LIN {X -0.120,Y -244.755,Z 514.218,A 0.000,B 0.000,C 90.000,E1 39.277} C_DIS
LIN {X -0.007,Y -235.366,Z 514.200,A 0.000,B 0.000,C 90.000,E1 35.931} C_DIS
LIN {X -0.130,Y -227.809,Z 514.183,A 0.000,B 0.000,C 90.000,E1 32.959} C_DIS
LIN {X 0.017,Y -221.054,Z 514.166,A 0.000,B 0.000,C 90.000,E1 29.873} C_DIS
LIN {X -0.038,Y -215.129,Z 514.149,A 0.000,B 0.000,C 90.000,E1 26.796} C_DIS
LIN {X 0.047,Y -210.062,Z 514.131,A 0.000,B 0.000,C 90.000,E1 23.643} C_DIS
LIN {X -0.028,Y -204.891,Z 514.109,A 0.000,B 0.000,C 90.000,E1 19.704} C_DIS
LIN {X -0.082,Y -200.758,Z 514.087,A 0.000,B 0.000,C 90.000,E1 15.717} C_DIS
LIN {X 0.030,Y -197.089,Z 514.060,A 0.000,B 0.000,C 90.000,E1 10.838} C_DIS
LIN {X -0.097,Y -194.452,Z 514.024,A 0.000,B 0.000,C 90.000,E1 4.359} C_DIS
LIN {X -0.009,Y -195.978,Z 513.961,A 0.000,B 0.000,C 90.000,E1 352.996} C_DIS
LIN {X 0.017,Y -199.614,Z 513.929,A 0.000,B 0.000,C 90.000,E1 347.297} C_DIS
LIN {X -0.001,Y -203.417,Z 513.907,A 0.000,B 0.000,C 90.000,E1 343.268} C_DIS
LIN {X 0.019,Y -208.024,Z 513.885,A 0.000,B 0.000,C 90.000,E1 339.263} C_DIS
LIN {X 0.017,Y -213.374,Z 513.863,A 0.000,B 0.000,C 90.000,E1 335.305} C_DIS
LIN {X 0.048,Y -219.357,Z 513.841,A 0.000,B 0.000,C 90.000,E1 331.385} C_DIS
LIN {X 0.009,Y -225.894,Z 513.820,A 0.000,B 0.000,C 90.000,E1 327.533} C_DIS
LIN {X 0.008,Y -231.651,Z 513.803,A 0.000,B 0.000,C 90.000,E1 324.482} C_DIS
LIN {X -0.005,Y -239.280,Z 513.782,A 0.000,B 0.000,C 90.000,E1 320.723} C_DIS
LIN {X -0.031,Y -247.836,Z 513.761,A 0.000,B 0.000,C 90.000,E1 317.025} C_DIS
LIN {X -0.010,Y -256.576,Z 513.743,A 0.000,B 0.000,C 90.000,E1 313.743} C_DIS
LIN {X 0.003,Y -267.396,Z 513.723,A 0.000,B 0.000,C 90.000,E1 310.172} C_DIS
LIN {X 0.088,Y -279.550,Z 513.704,A 0.000,B 0.000,C 90.000,E1 306.664} C_DIS
LIN {X -0.111,Y -292.992,Z 513.685,A 0.000,B 0.000,C 90.000,E1 303.293} C_DIS
LIN {X 0.095,Y -305.926,Z 513.668,A 0.000,B 0.000,C 90.000,E1 300.256} C_DIS
LIN {X 0.147,Y -321.556,Z 513.650,A 0.000,B 0.000,C 90.000,E1 297.001} C_DIS
LIN {X -0.195,Y -332.000,Z 513.640,A 0.000,B 0.000,C 90.000,E1 295.155} C_DIS
LIN {X -0.025,Y -349.412,Z 513.624,A 0.000,B 0.000,C 90.000,E1 292.333} C_DIS
LIN {X -0.077,Y -368.920,Z 513.609,A 0.000,B 0.000,C 90.000,E1 289.631} C_DIS
LIN {X 0.072,Y -390.367,Z 513.594,A 0.000,B 0.000,C 90.000,E1 286.985} C_DIS
LIN {X -0.161,Y -412.698,Z 513.580,A 0.000,B 0.000,C 90.000,E1 284.481} C_DIS
LIN {X 0.197,Y -425.211,Z 513.573,A 0.000,B 0.000,C 90.000,E1 283.063} C_DIS
LIN {X -0.216,Y -437.299,Z 513.565,A 0.000,B 0.000,C 90.000,E1 281.771} C_DIS
LIN {X 0.182,Y -446.567,Z 513.559,A 0.000,B 0.000,C 90.000,E1 280.658} C_DIS
LIN {X 0.176,Y -455.192,Z 513.554,A 0.000,B 0.000,C 90.000,E1 279.613} C_DIS
LIN {X -0.004,Y -461.099,Z 513.549,A 0.000,B 0.000,C 90.000,E1 278.859} C_DIS
LIN {X -0.140,Y -466.456,Z 513.545,A 0.000,B 0.000,C 90.000,E1 278.106} C_DIS
LIN {X 0.240,Y -471.291,Z 513.541,A 0.000,B 0.000,C 90.000,E1 277.296} C_DIS
LIN {X 0.136,Y -475.580,Z 513.536,A 0.000,B 0.000,C 90.000,E1 276.549} C_DIS
LIN {X 0.127,Y -479.382,Z 513.532,A 0.000,B 0.000,C 90.000,E1 275.796} C_DIS
LIN {X 0.096,Y -482.574,Z 513.528,A 0.000,B 0.000,C 90.000,E1 275.049} C_DIS
LIN {X -0.215,Y -484.338,Z 513.525,A 0.000,B 0.000,C 90.000,E1 274.588} C_DIS
LIN {X -0.075,Y -485.711,Z 513.523,A 0.000,B 0.000,C 90.000,E1 274.073} C_DIS
LIN {X 0.111,Y -486.806,Z 513.520,A 0.000,B 0.000,C 90.000,E1 273.555} C_DIS
LIN {X -0.185,Y -487.563,Z 513.517,A 0.000,B 0.000,C 90.000,E1 273.094} C_DIS
LIN {X -0.013,Y -487.993,Z 513.514,A 0.000,B 0.000,C 90.000,E1 272.579} C_DIS
LIN {X 0.165,Y -487.997,Z 513.512,A 0.000,B 0.000,C 90.000,E1 272.064} C_DIS
LIN {X -0.126,Y -487.649,Z 513.509,A 0.000,B 0.000,C 90.000,E1 271.604} C_DIS
LIN {X 0.056,Y -486.936,Z 513.506,A 0.000,B 0.000,C 90.000,E1 271.088} C_DIS
LIN {X 0.236,Y -485.739,Z 513.503,A 0.000,B 0.000,C 90.000,E1 270.573} C_DIS
LIN {X -0.073,Y -483.979,Z 513.501,A 0.000,B 0.000,C 90.000,E1 270.115} C_DIS
LIN {X 0.096,Y -481.572,Z 513.498,A 0.000,B 0.000,C 90.000,E1 269.599} C_DIS
LIN {X -0.232,Y -478.454,Z 513.495,A 0.000,B 0.000,C 90.000,E1 269.141} C_DIS
LIN {X -0.097,Y -474.407,Z 513.492,A 0.000,B 0.000,C 90.000,E1 268.625} C_DIS
LIN {X 0.195,Y -472.055,Z 513.491,A 0.000,B 0.000,C 90.000,E1 268.339} C_DIS
LIN {X -0.019,Y -466.542,Z 513.488,A 0.000,B 0.000,C 90.000,E1 267.879} C_DIS
LIN {X 0.146,Y -460.305,Z 513.486,A 0.000,B 0.000,C 90.000,E1 267.421} C_DIS
LIN {X -0.101,Y -456.798,Z 513.485,A 0.000,B 0.000,C 90.000,E1 267.249} C_DIS
LIN {X -0.038,Y -449.866,Z 513.483,A 0.000,B 0.000,C 90.000,E1 266.906} C_DIS
LIN {X 0.031,Y -442.828,Z 513.481,A 0.000,B 0.000,C 90.000,E1 266.617} C_DIS
LIN {X -0.015,Y -435.647,Z 513.480,A 0.000,B 0.000,C 90.000,E1 266.388} C_DIS
LIN {X -0.171,Y -427.820,Z 513.479,A 0.000,B 0.000,C 90.000,E1 266.216} C_DIS
LIN {X 0.052,Y -417.909,Z 513.478,A 0.000,B 0.000,C 90.000,E1 266.045} C_DIS
LIN {X 0.067,Y -409.310,Z 513.478,A 0.000,B 0.000,C 90.000,E1 265.988} C_DIS
LIN {X -0.005,Y -180.920,Z 513.478,A 0.000,B 0.000,C 90.000,E1 265.988} C_DIS
LIN {X -0.002,Y -180.885,Z 513.473,A 0.000,B 0.000,C 90.000,E1 265.122} C_DIS
LIN {X 0.056,Y -179.006,Z 513.445,A 0.000,B 0.000,C 90.000,E1 260.038} C_DIS
LIN {X -0.025,Y -178.614,Z 513.440,A 0.000,B 0.000,C 90.000,E1 259.218} C_DIS
LIN {X 0.043,Y -175.665,Z 513.412,A 0.000,B 0.000,C 90.000,E1 254.102} C_DIS
LIN {X 0.048,Y -172.383,Z 513.388,A 0.000,B 0.000,C 90.000,E1 249.826} C_DIS
LIN {X 0.062,Y -171.183,Z 513.378,A 0.000,B 0.000,C 90.000,E1 248.103} C_DIS
LIN {X -0.045,Y -167.476,Z 513.354,A 0.000,B 0.000,C 90.000,E1 243.819} C_DIS
LIN {X 0.039,Y -166.872,Z 513.350,A 0.000,B 0.000,C 90.000,E1 242.922} C_DIS
LIN {X -0.045,Y -162.177,Z 513.320,A 0.000,B 0.000,C 90.000,E1 237.709} C_DIS
LIN {X 0.013,Y -160.742,Z 513.311,A 0.000,B 0.000,C 90.000,E1 235.928} C_DIS
LIN {X -0.008,Y -157.542,Z 513.291,A 0.000,B 0.000,C 90.000,E1 232.396} C_DIS
LIN {X 0.048,Y -155.570,Z 513.276,A 0.000,B 0.000,C 90.000,E1 229.703} C_DIS
LIN {X -0.019,Y -151.857,Z 513.251,A 0.000,B 0.000,C 90.000,E1 225.243} C_DIS
LIN {X -0.004,Y -150.079,Z 513.236,A 0.000,B 0.000,C 90.000,E1 222.528} C_DIS
LIN {X 0.030,Y -146.884,Z 513.211,A 0.000,B 0.000,C 90.000,E1 217.971} C_DIS
LIN {X 0.019,Y -145.470,Z 513.196,A 0.000,B 0.000,C 90.000,E1 215.231} C_DIS
LIN {X -0.064,Y -142.882,Z 513.170,A 0.000,B 0.000,C 90.000,E1 210.669} C_DIS
LIN {X -0.007,Y -141.501,Z 513.150,A 0.000,B 0.000,C 90.000,E1 206.950} C_DIS
LIN {X 0.042,Y -139.388,Z 513.114,A 0.000,B 0.000,C 90.000,E1 200.429} C_DIS
LIN {X 0.030,Y -138.845,Z 513.098,A 0.000,B 0.000,C 90.000,E1 197.638} C_DIS
LIN {X -0.046,Y -138.353,Z 513.057,A 0.000,B 0.000,C 90.000,E1 190.197} C_DIS
LIN {X -0.054,Y -139.517,Z 513.005,A 0.000,B 0.000,C 90.000,E1 180.859} C_DIS
LIN {X 0.027,Y -141.172,Z 512.974,A 0.000,B 0.000,C 90.000,E1 175.241} C_DIS
LIN {X -0.002,Y -142.552,Z 512.958,A 0.000,B 0.000,C 90.000,E1 172.470} C_DIS
LIN {X -0.076,Y -144.830,Z 512.932,A 0.000,B 0.000,C 90.000,E1 167.881} C_DIS
LIN {X 0.052,Y -147.452,Z 512.912,A 0.000,B 0.000,C 90.000,E1 164.157} C_DIS
LIN {X -0.062,Y -150.033,Z 512.892,A 0.000,B 0.000,C 90.000,E1 160.550} C_DIS
LIN {X -0.056,Y -153.372,Z 512.872,A 0.000,B 0.000,C 90.000,E1 156.922} C_DIS
LIN {X -0.008,Y -155.905,Z 512.857,A 0.000,B 0.000,C 90.000,E1 154.204} C_DIS
LIN {X -0.032,Y -159.766,Z 512.837,A 0.000,B 0.000,C 90.000,E1 150.639} C_DIS
LIN {X -0.045,Y -162.006,Z 512.827,A 0.000,B 0.000,C 90.000,E1 148.869} C_DIS
LIN {X 0.069,Y -166.199,Z 512.807,A 0.000,B 0.000,C 90.000,E1 145.308} C_DIS
LIN {X 0.072,Y -171.215,Z 512.788,A 0.000,B 0.000,C 90.000,E1 141.823} C_DIS
LIN {X -0.005,Y -176.099,Z 512.769,A 0.000,B 0.000,C 90.000,E1 138.405} C_DIS
LIN {X 0.113,Y -180.362,Z 512.755,A 0.000,B 0.000,C 90.000,E1 135.810} C_DIS
LIN {X 0.090,Y -185.771,Z 512.736,A 0.000,B 0.000,C 90.000,E1 132.447} C_DIS
LIN {X 0.023,Y -190.385,Z 512.722,A 0.000,B 0.000,C 90.000,E1 129.967} C_DIS
LIN {X 0.020,Y -192.445,Z 512.715,A 0.000,B 0.000,C 90.000,E1 128.749} C_DIS
LIN {X -0.013,Y -289.228,Z 512.715,A 0.000,B 0.000,C 90.000,E1 128.749} C_DIS
LIN {X -0.057,Y -290.139,Z 512.715,A 0.000,B 0.000,C 90.000,E1 128.749} C_DIS
LIN {X -0.072,Y -295.347,Z 512.714,A 0.000,B 0.000,C 90.000,E1 128.543} C_DIS
LIN {X 0.100,Y -297.889,Z 512.713,A 0.000,B 0.000,C 90.000,E1 128.302} C_DIS
LIN {X 0.151,Y -301.704,Z 512.710,A 0.000,B 0.000,C 90.000,E1 127.810} C_DIS
LIN {X -0.090,Y -303.526,Z 512.708,A 0.000,B 0.000,C 90.000,E1 127.523} C_DIS
LIN {X 0.094,Y -304.951,Z 512.707,A 0.000,B 0.000,C 90.000,E1 127.156} C_DIS
LIN {X 0.071,Y -306.993,Z 512.703,A 0.000,B 0.000,C 90.000,E1 126.503} C_DIS
LIN {X 0.104,Y -317.017,Z 512.685,A 0.000,B 0.000,C 90.000,E1 123.245} C_DIS
LIN {X 0.027,Y -327.358,Z 512.669,A 0.000,B 0.000,C 90.000,E1 120.384} C_DIS
LIN {X -0.142,Y -339.055,Z 512.653,A 0.000,B 0.000,C 90.000,E1 117.590} C_DIS
LIN {X 0.187,Y -352.208,Z 512.638,A 0.000,B 0.000,C 90.000,E1 114.771} C_DIS
LIN {X 0.056,Y -365.222,Z 512.624,A 0.000,B 0.000,C 90.000,E1 112.386} C_DIS
LIN {X -0.172,Y -379.577,Z 512.611,A 0.000,B 0.000,C 90.000,E1 110.066} C_DIS
LIN {X -0.168,Y -395.376,Z 512.599,A 0.000,B 0.000,C 90.000,E1 107.764} C_DIS
LIN {X 0.109,Y -412.737,Z 512.586,A 0.000,B 0.000,C 90.000,E1 105.481} C_DIS
LIN {X 0.108,Y -431.774,Z 512.574,A 0.000,B 0.000,C 90.000,E1 103.300} C_DIS
LIN {X 0.167,Y -451.899,Z 512.563,A 0.000,B 0.000,C 90.000,E1 101.243} C_DIS
LIN {X 0.055,Y -472.572,Z 512.552,A 0.000,B 0.000,C 90.000,E1 99.378} C_DIS
LIN {X 0.192,Y -477.818,Z 512.550,A 0.000,B 0.000,C 90.000,E1 98.916} C_DIS
LIN {X -0.229,Y -480.089,Z 512.548,A 0.000,B 0.000,C 90.000,E1 98.746} C_DIS
LIN {X 0.198,Y -481.950,Z 512.547,A 0.000,B 0.000,C 90.000,E1 98.454} C_DIS
LIN {X 0.149,Y -483.362,Z 512.546,A 0.000,B 0.000,C 90.000,E1 98.219} C_DIS
LIN {X -0.159,Y -485.241,Z 512.543,A 0.000,B 0.000,C 90.000,E1 97.757} C_DIS
LIN {X 0.023,Y -486.010,Z 512.540,A 0.000,B 0.000,C 90.000,E1 97.239} C_DIS
LIN {X 0.218,Y -485.794,Z 512.537,A 0.000,B 0.000,C 90.000,E1 96.720} C_DIS
LIN {X -0.066,Y -484.563,Z 512.535,A 0.000,B 0.000,C 90.000,E1 96.258} C_DIS
LIN {X -0.182,Y -483.507,Z 512.533,A 0.000,B 0.000,C 90.000,E1 96.024} C_DIS
LIN {X 0.131,Y -482.084,Z 512.532,A 0.000,B 0.000,C 90.000,E1 95.739} C_DIS
LIN {X -0.005,Y -474.162,Z 512.526,A 0.000,B 0.000,C 90.000,E1 94.759} C_DIS
LIN {X 0.071,Y -460.399,Z 512.517,A 0.000,B 0.000,C 90.000,E1 92.980} C_DIS
LIN {X -0.110,Y -451.472,Z 512.509,A 0.000,B 0.000,C 90.000,E1 91.718} C_DIS
LIN {X -0.135,Y -436.900,Z 512.496,A 0.000,B 0.000,C 90.000,E1 89.370} C_DIS
LIN {X 0.203,Y -423.873,Z 512.485,A 0.000,B 0.000,C 90.000,E1 87.192} C_DIS
LIN {X -0.138,Y -411.086,Z 512.472,A 0.000,B 0.000,C 90.000,E1 85.065} C_DIS
LIN {X 0.117,Y -397.019,Z 512.459,A 0.000,B 0.000,C 90.000,E1 82.534} C_DIS
LIN {X 0.107,Y -386.038,Z 512.448,A 0.000,B 0.000,C 90.000,E1 80.557} C_DIS
LIN {X -0.111,Y -375.042,Z 512.436,A 0.000,B 0.000,C 90.000,E1 78.578} C_DIS
LIN {X -0.045,Y -364.309,Z 512.425,A 0.000,B 0.000,C 90.000,E1 76.520} C_DIS
LIN {X -0.165,Y -353.218,Z 512.412,A 0.000,B 0.000,C 90.000,E1 74.157} C_DIS
LIN {X 0.067,Y -344.586,Z 512.400,A 0.000,B 0.000,C 90.000,E1 72.000} C_DIS
LIN {X -0.120,Y -333.650,Z 512.383,A 0.000,B 0.000,C 90.000,E1 68.954} C_DIS
LIN {X -0.035,Y -321.585,Z 512.362,A 0.000,B 0.000,C 90.000,E1 65.177} C_DIS
LIN {X 0.020,Y -313.768,Z 512.348,A 0.000,B 0.000,C 90.000,E1 62.615} C_DIS
LIN {X 0.077,Y -307.963,Z 512.337,A 0.000,B 0.000,C 90.000,E1 60.667} C_DIS
LIN {X -0.032,Y -300.214,Z 512.323,A 0.000,B 0.000,C 90.000,E1 58.074} C_DIS
LIN {X -0.101,Y -290.942,Z 512.304,A 0.000,B 0.000,C 90.000,E1 54.769} C_DIS
LIN {X -0.055,Y -283.932,Z 512.289,A 0.000,B 0.000,C 90.000,E1 52.065} C_DIS
LIN {X -0.147,Y -280.320,Z 512.282,A 0.000,B 0.000,C 90.000,E1 50.723} C_DIS
LIN {X -0.061,Y -274.511,Z 512.270,A 0.000,B 0.000,C 90.000,E1 48.647} C_DIS
LIN {X -0.018,Y -269.212,Z 512.261,A 0.000,B 0.000,C 90.000,E1 46.905} C_DIS
LIN {X -0.009,Y -262.316,Z 512.249,A 0.000,B 0.000,C 90.000,E1 44.798} C_DIS
LIN {X -0.058,Y -251.867,Z 512.231,A 0.000,B 0.000,C 90.000,E1 41.595} C_DIS
LIN {X 0.008,Y -242.993,Z 512.215,A 0.000,B 0.000,C 90.000,E1 38.669} C_DIS
LIN {X -0.042,Y -234.757,Z 512.198,A 0.000,B 0.000,C 90.000,E1 35.724} C_DIS
LIN {X 0.014,Y -227.236,Z 512.182,A 0.000,B 0.000,C 90.000,E1 32.704} C_DIS
LIN {X -0.045,Y -220.548,Z 512.165,A 0.000,B 0.000,C 90.000,E1 29.667} C_DIS
LIN {X -0.019,Y -214.687,Z 512.148,A 0.000,B 0.000,C 90.000,E1 26.565} C_DIS
LIN {X -0.045,Y -209.696,Z 512.130,A 0.000,B 0.000,C 90.000,E1 23.439} C_DIS
LIN {X 0.055,Y -204.595,Z 512.108,A 0.000,B 0.000,C 90.000,E1 19.450} C_DIS
LIN {X -0.074,Y -200.511,Z 512.086,A 0.000,B 0.000,C 90.000,E1 15.481} C_DIS
LIN {X 0.028,Y -196.901,Z 512.059,A 0.000,B 0.000,C 90.000,E1 10.602} C_DIS
LIN {X 0.063,Y -194.347,Z 512.023,A 0.000,B 0.000,C 90.000,E1 4.073} C_DIS
LIN {X -0.014,Y -195.866,Z 511.961,A 0.000,B 0.000,C 90.000,E1 352.996} C_DIS
LIN {X 0.006,Y -199.485,Z 511.929,A 0.000,B 0.000,C 90.000,E1 347.297} C_DIS
LIN {X -0.016,Y -203.277,Z 511.907,A 0.000,B 0.000,C 90.000,E1 343.268} C_DIS
LIN {X -0.001,Y -207.891,Z 511.885,A 0.000,B 0.000,C 90.000,E1 339.263} C_DIS
LIN {X -0.007,Y -213.248,Z 511.863,A 0.000,B 0.000,C 90.000,E1 335.305} C_DIS
LIN {X 0.019,Y -219.221,Z 511.841,A 0.000,B 0.000,C 90.000,E1 331.385} C_DIS
LIN {X -0.026,Y -225.768,Z 511.820,A 0.000,B 0.000,C 90.000,E1 327.533} C_DIS
LIN {X -0.030,Y -231.544,Z 511.803,A 0.000,B 0.000,C 90.000,E1 324.482} C_DIS
LIN {X -0.047,Y -239.189,Z 511.782,A 0.000,B 0.000,C 90.000,E1 320.723} C_DIS
LIN {X 0.091,Y -247.765,Z 511.761,A 0.000,B 0.000,C 90.000,E1 316.986} C_DIS
LIN {X -0.048,Y -257.577,Z 511.741,A 0.000,B 0.000,C 90.000,E1 313.380} C_DIS
LIN {X 0.013,Y -268.530,Z 511.721,A 0.000,B 0.000,C 90.000,E1 309.806} C_DIS
LIN {X 0.135,Y -280.829,Z 511.702,A 0.000,B 0.000,C 90.000,E1 306.297} C_DIS
LIN {X -0.188,Y -294.405,Z 511.683,A 0.000,B 0.000,C 90.000,E1 302.959} C_DIS
LIN {X -0.060,Y -308.915,Z 511.664,A 0.000,B 0.000,C 90.000,E1 299.617} C_DIS
LIN {X 0.014,Y -323.243,Z 511.648,A 0.000,B 0.000,C 90.000,E1 296.693} C_DIS
LIN {X 0.146,Y -333.874,Z 511.638,A 0.000,B 0.000,C 90.000,E1 294.771} C_DIS
LIN {X -0.095,Y -349.446,Z 511.624,A 0.000,B 0.000,C 90.000,E1 292.333} C_DIS
LIN {X -0.152,Y -368.953,Z 511.609,A 0.000,B 0.000,C 90.000,E1 289.631} C_DIS
LIN {X -0.005,Y -390.388,Z 511.594,A 0.000,B 0.000,C 90.000,E1 286.985} C_DIS
LIN {X -0.197,Y -412.721,Z 511.580,A 0.000,B 0.000,C 90.000,E1 284.481} C_DIS
LIN {X -0.138,Y -425.120,Z 511.573,A 0.000,B 0.000,C 90.000,E1 283.119} C_DIS
LIN {X -0.135,Y -437.238,Z 511.565,A 0.000,B 0.000,C 90.000,E1 281.771} C_DIS
LIN {X -0.175,Y -446.550,Z 511.559,A 0.000,B 0.000,C 90.000,E1 280.715} C_DIS
LIN {X 0.011,Y -453.120,Z 511.555,A 0.000,B 0.000,C 90.000,E1 279.905} C_DIS
LIN {X -0.194,Y -459.252,Z 511.551,A 0.000,B 0.000,C 90.000,E1 279.151} C_DIS
LIN {X 0.119,Y -464.777,Z 511.546,A 0.000,B 0.000,C 90.000,E1 278.341} C_DIS
LIN {X 0.017,Y -469.791,Z 511.542,A 0.000,B 0.000,C 90.000,E1 277.587} C_DIS
LIN {X -0.041,Y -474.245,Z 511.538,A 0.000,B 0.000,C 90.000,E1 276.834} C_DIS
LIN {X -0.119,Y -478.215,Z 511.534,A 0.000,B 0.000,C 90.000,E1 276.087} C_DIS
LIN {X -0.111,Y -481.656,Z 511.530,A 0.000,B 0.000,C 90.000,E1 275.334} C_DIS
LIN {X -0.124,Y -484.402,Z 511.525,A 0.000,B 0.000,C 90.000,E1 274.588} C_DIS
LIN {X 0.017,Y -485.820,Z 511.523,A 0.000,B 0.000,C 90.000,E1 274.073} C_DIS
LIN {X 0.204,Y -486.894,Z 511.520,A 0.000,B 0.000,C 90.000,E1 273.555} C_DIS
LIN {X -0.091,Y -487.670,Z 511.517,A 0.000,B 0.000,C 90.000,E1 273.094} C_DIS
LIN {X 0.080,Y -488.091,Z 511.514,A 0.000,B 0.000,C 90.000,E1 272.579} C_DIS
LIN {X -0.228,Y -488.143,Z 511.512,A 0.000,B 0.000,C 90.000,E1 272.121} C_DIS
LIN {X -0.030,Y -487.800,Z 511.509,A 0.000,B 0.000,C 90.000,E1 271.604} C_DIS
LIN {X 0.152,Y -487.051,Z 511.506,A 0.000,B 0.000,C 90.000,E1 271.088} C_DIS
LIN {X -0.153,Y -485.877,Z 511.503,A 0.000,B 0.000,C 90.000,E1 270.630} C_DIS
LIN {X 0.024,Y -484.136,Z 511.501,A 0.000,B 0.000,C 90.000,E1 270.115} C_DIS
LIN {X 0.193,Y -481.736,Z 511.498,A 0.000,B 0.000,C 90.000,E1 269.599} C_DIS
LIN {X -0.135,Y -478.606,Z 511.495,A 0.000,B 0.000,C 90.000,E1 269.141} C_DIS
LIN {X 0.001,Y -474.582,Z 511.492,A 0.000,B 0.000,C 90.000,E1 268.625} C_DIS
LIN {X -0.180,Y -472.222,Z 511.491,A 0.000,B 0.000,C 90.000,E1 268.396} C_DIS
LIN {X 0.054,Y -466.727,Z 511.488,A 0.000,B 0.000,C 90.000,E1 267.879} C_DIS
LIN {X 0.189,Y -460.442,Z 511.486,A 0.000,B 0.000,C 90.000,E1 267.421} C_DIS
LIN {X -0.028,Y -453.674,Z 511.484,A 0.000,B 0.000,C 90.000,E1 267.078} C_DIS
LIN {X -0.160,Y -446.790,Z 511.482,A 0.000,B 0.000,C 90.000,E1 266.788} C_DIS
LIN {X 0.047,Y -439.832,Z 511.481,A 0.000,B 0.000,C 90.000,E1 266.502} C_DIS
LIN {X 0.133,Y -432.419,Z 511.479,A 0.000,B 0.000,C 90.000,E1 266.274} C_DIS
LIN {X 0.152,Y -423.889,Z 511.478,A 0.000,B 0.000,C 90.000,E1 266.102} C_DIS
LIN {X 0.044,Y -418.120,Z 511.478,A 0.000,B 0.000,C 90.000,E1 266.045} C_DIS
LIN {X 0.058,Y -410.283,Z 511.478,A 0.000,B 0.000,C 90.000,E1 265.988} C_DIS
LIN {X -0.009,Y -180.919,Z 511.478,A 0.000,B 0.000,C 90.000,E1 265.988} C_DIS
LIN {X -0.007,Y -180.885,Z 511.473,A 0.000,B 0.000,C 90.000,E1 265.122} C_DIS
LIN {X 0.052,Y -179.006,Z 511.445,A 0.000,B 0.000,C 90.000,E1 260.038} C_DIS
LIN {X -0.029,Y -178.612,Z 511.440,A 0.000,B 0.000,C 90.000,E1 259.218} C_DIS
LIN {X 0.039,Y -175.664,Z 511.412,A 0.000,B 0.000,C 90.000,E1 254.102} C_DIS
LIN {X 0.044,Y -172.382,Z 511.388,A 0.000,B 0.000,C 90.000,E1 249.826} C_DIS
LIN {X 0.058,Y -171.181,Z 511.378,A 0.000,B 0.000,C 90.000,E1 248.103} C_DIS
LIN {X -0.049,Y -167.475,Z 511.354,A 0.000,B 0.000,C 90.000,E1 243.819} C_DIS
LIN {X 0.034,Y -166.871,Z 511.350,A 0.000,B 0.000,C 90.000,E1 242.922} C_DIS
LIN {X -0.049,Y -162.176,Z 511.320,A 0.000,B 0.000,C 90.000,E1 237.709} C_DIS
LIN {X 0.008,Y -160.741,Z 511.311,A 0.000,B 0.000,C 90.000,E1 235.928} C_DIS
LIN {X -0.013,Y -157.542,Z 511.291,A 0.000,B 0.000,C 90.000,E1 232.396} C_DIS
LIN {X 0.045,Y -155.569,Z 511.276,A 0.000,B 0.000,C 90.000,E1 229.703} C_DIS
LIN {X -0.022,Y -151.857,Z 511.251,A 0.000,B 0.000,C 90.000,E1 225.243} C_DIS
LIN {X -0.008,Y -150.078,Z 511.236,A 0.000,B 0.000,C 90.000,E1 222.528} C_DIS
LIN {X 0.026,Y -146.883,Z 511.211,A 0.000,B 0.000,C 90.000,E1 217.971} C_DIS
LIN {X 0.015,Y -145.469,Z 511.196,A 0.000,B 0.000,C 90.000,E1 215.231} C_DIS
LIN {X -0.068,Y -142.881,Z 511.170,A 0.000,B 0.000,C 90.000,E1 210.669} C_DIS
LIN {X -0.011,Y -141.500,Z 511.150,A 0.000,B 0.000,C 90.000,E1 206.950} C_DIS
LIN {X 0.038,Y -139.387,Z 511.114,A 0.000,B 0.000,C 90.000,E1 200.429} C_DIS
LIN {X 0.027,Y -138.845,Z 511.098,A 0.000,B 0.000,C 90.000,E1 197.638} C_DIS
LIN {X -0.049,Y -138.354,Z 511.057,A 0.000,B 0.000,C 90.000,E1 190.197} C_DIS
LIN {X -0.058,Y -139.517,Z 511.005,A 0.000,B 0.000,C 90.000,E1 180.859} C_DIS
LIN {X 0.023,Y -141.174,Z 510.974,A 0.000,B 0.000,C 90.000,E1 175.241} C_DIS
LIN {X -0.006,Y -142.552,Z 510.958,A 0.000,B 0.000,C 90.000,E1 172.470} C_DIS
LIN {X -0.080,Y -144.830,Z 510.932,A 0.000,B 0.000,C 90.000,E1 167.881} C_DIS
LIN {X 0.048,Y -147.453,Z 510.912,A 0.000,B 0.000,C 90.000,E1 164.157} C_DIS
LIN {X -0.066,Y -150.035,Z 510.892,A 0.000,B 0.000,C 90.000,E1 160.550} C_DIS
LIN {X -0.060,Y -153.374,Z 510.872,A 0.000,B 0.000,C 90.000,E1 156.922} C_DIS
LIN {X -0.012,Y -155.906,Z 510.857,A 0.000,B 0.000,C 90.000,E1 154.204} C_DIS
LIN {X 0.103,Y -159.768,Z 510.837,A 0.000,B 0.000,C 90.000,E1 150.589} C_DIS
LIN {X -0.049,Y -162.008,Z 510.827,A 0.000,B 0.000,C 90.000,E1 148.869} C_DIS
LIN {X 0.064,Y -166.201,Z 510.807,A 0.000,B 0.000,C 90.000,E1 145.308} C_DIS
LIN {X 0.067,Y -171.217,Z 510.788,A 0.000,B 0.000,C 90.000,E1 141.823} C_DIS
LIN {X -0.009,Y -176.102,Z 510.769,A 0.000,B 0.000,C 90.000,E1 138.405} C_DIS
LIN {X 0.108,Y -180.364,Z 510.755,A 0.000,B 0.000,C 90.000,E1 135.810} C_DIS
LIN {X 0.086,Y -185.773,Z 510.736,A 0.000,B 0.000,C 90.000,E1 132.447} C_DIS
LIN {X 0.018,Y -190.388,Z 510.722,A 0.000,B 0.000,C 90.000,E1 129.967} C_DIS
LIN {X -0.091,Y -192.501,Z 510.715,A 0.000,B 0.000,C 90.000,E1 128.749} C_DIS
LIN {X 0.055,Y -289.106,Z 510.715,A 0.000,B 0.000,C 90.000,E1 128.705} C_DIS
LIN {X 0.063,Y -291.444,Z 510.715,A 0.000,B 0.000,C 90.000,E1 128.669} C_DIS
LIN {X -0.038,Y -295.372,Z 510.714,A 0.000,B 0.000,C 90.000,E1 128.508} C_DIS
LIN {X 0.093,Y -297.636,Z 510.713,A 0.000,B 0.000,C 90.000,E1 128.302} C_DIS
LIN {X -0.035,Y -301.507,Z 510.710,A 0.000,B 0.000,C 90.000,E1 127.855} C_DIS
LIN {X -0.020,Y -303.372,Z 510.708,A 0.000,B 0.000,C 90.000,E1 127.523} C_DIS
LIN {X 0.181,Y -304.833,Z 510.707,A 0.000,B 0.000,C 90.000,E1 127.156} C_DIS
LIN {X 0.159,Y -306.927,Z 510.703,A 0.000,B 0.000,C 90.000,E1 126.503} C_DIS
LIN {X -0.074,Y -316.942,Z 510.685,A 0.000,B 0.000,C 90.000,E1 123.293} C_DIS
LIN {X -0.050,Y -327.277,Z 510.669,A 0.000,B 0.000,C 90.000,E1 120.413} C_DIS
LIN {X -0.053,Y -338.966,Z 510.653,A 0.000,B 0.000,C 90.000,E1 117.590} C_DIS
LIN {X -0.042,Y -352.110,Z 510.638,A 0.000,B 0.000,C 90.000,E1 114.823} C_DIS
LIN {X 0.008,Y -365.117,Z 510.625,A 0.000,B 0.000,C 90.000,E1 112.408} C_DIS
LIN {X -0.080,Y -379.461,Z 510.611,A 0.000,B 0.000,C 90.000,E1 110.066} C_DIS
LIN {X -0.075,Y -395.253,Z 510.599,A 0.000,B 0.000,C 90.000,E1 107.764} C_DIS
LIN {X 0.204,Y -412.603,Z 510.586,A 0.000,B 0.000,C 90.000,E1 105.481} C_DIS
LIN {X 0.201,Y -431.630,Z 510.574,A 0.000,B 0.000,C 90.000,E1 103.300} C_DIS
LIN {X -0.187,Y -451.753,Z 510.563,A 0.000,B 0.000,C 90.000,E1 101.299} C_DIS
LIN {X 0.139,Y -472.423,Z 510.552,A 0.000,B 0.000,C 90.000,E1 99.378} C_DIS
LIN {X -0.196,Y -477.668,Z 510.550,A 0.000,B 0.000,C 90.000,E1 98.973} C_DIS
LIN {X -0.146,Y -480.018,Z 510.548,A 0.000,B 0.000,C 90.000,E1 98.746} C_DIS
LIN {X -0.154,Y -481.904,Z 510.547,A 0.000,B 0.000,C 90.000,E1 98.511} C_DIS
LIN {X -0.164,Y -483.342,Z 510.546,A 0.000,B 0.000,C 90.000,E1 98.276} C_DIS
LIN {X 0.008,Y -485.313,Z 510.543,A 0.000,B 0.000,C 90.000,E1 97.757} C_DIS
LIN {X 0.190,Y -486.155,Z 510.540,A 0.000,B 0.000,C 90.000,E1 97.239} C_DIS
LIN {X -0.098,Y -486.009,Z 510.538,A 0.000,B 0.000,C 90.000,E1 96.777} C_DIS
LIN {X 0.102,Y -484.856,Z 510.535,A 0.000,B 0.000,C 90.000,E1 96.258} C_DIS
LIN {X -0.065,Y -483.846,Z 510.533,A 0.000,B 0.000,C 90.000,E1 96.030} C_DIS
LIN {X -0.181,Y -482.481,Z 510.532,A 0.000,B 0.000,C 90.000,E1 95.796} C_DIS
LIN {X 0.003,Y -478.668,Z 510.529,A 0.000,B 0.000,C 90.000,E1 95.277} C_DIS
LIN {X -0.216,Y -460.814,Z 510.517,A 0.000,B 0.000,C 90.000,E1 93.037} C_DIS
LIN {X 0.065,Y -451.837,Z 510.510,A 0.000,B 0.000,C 90.000,E1 91.718} C_DIS
LIN {X 0.043,Y -437.213,Z 510.497,A 0.000,B 0.000,C 90.000,E1 89.370} C_DIS
LIN {X -0.040,Y -424.180,Z 510.485,A 0.000,B 0.000,C 90.000,E1 87.249} C_DIS
LIN {X 0.045,Y -411.362,Z 510.473,A 0.000,B 0.000,C 90.000,E1 85.065} C_DIS
LIN {X -0.093,Y -397.286,Z 510.459,A 0.000,B 0.000,C 90.000,E1 82.591} C_DIS
LIN {X -0.152,Y -386.312,Z 510.448,A 0.000,B 0.000,C 90.000,E1 80.622} C_DIS
LIN {X 0.074,Y -375.305,Z 510.437,A 0.000,B 0.000,C 90.000,E1 78.578} C_DIS
LIN {X 0.055,Y -364.562,Z 510.425,A 0.000,B 0.000,C 90.000,E1 76.533} C_DIS
LIN {X 0.021,Y -353.443,Z 510.412,A 0.000,B 0.000,C 90.000,E1 74.157} C_DIS
LIN {X -0.099,Y -345.947,Z 510.402,A 0.000,B 0.000,C 90.000,E1 72.362} C_DIS
LIN {X 0.034,Y -331.676,Z 510.380,A 0.000,B 0.000,C 90.000,E1 68.337} C_DIS
LIN {X -0.150,Y -321.683,Z 510.362,A 0.000,B 0.000,C 90.000,E1 65.229} C_DIS
LIN {X -0.085,Y -313.862,Z 510.348,A 0.000,B 0.000,C 90.000,E1 62.666} C_DIS
LIN {X -0.018,Y -308.033,Z 510.337,A 0.000,B 0.000,C 90.000,E1 60.717} C_DIS
LIN {X -0.116,Y -300.256,Z 510.323,A 0.000,B 0.000,C 90.000,E1 58.122} C_DIS
LIN {X 0.066,Y -290.958,Z 510.304,A 0.000,B 0.000,C 90.000,E1 54.769} C_DIS
LIN {X -0.117,Y -283.934,Z 510.289,A 0.000,B 0.000,C 90.000,E1 52.110} C_DIS
LIN {X 0.013,Y -280.329,Z 510.282,A 0.000,B 0.000,C 90.000,E1 50.723} C_DIS
LIN {X -0.110,Y -274.531,Z 510.270,A 0.000,B 0.000,C 90.000,E1 48.690} C_DIS
LIN {X -0.047,Y -269.231,Z 510.261,A 0.000,B 0.000,C 90.000,E1 46.944} C_DIS
LIN {X -0.044,Y -262.323,Z 510.249,A 0.000,B 0.000,C 90.000,E1 44.838} C_DIS
LIN {X -0.109,Y -253.025,Z 510.233,A 0.000,B 0.000,C 90.000,E1 42.000} C_DIS
LIN {X -0.002,Y -243.046,Z 510.215,A 0.000,B 0.000,C 90.000,E1 38.705} C_DIS
LIN {X 0.096,Y -234.808,Z 510.199,A 0.000,B 0.000,C 90.000,E1 35.724} C_DIS
LIN {X -0.044,Y -227.258,Z 510.182,A 0.000,B 0.000,C 90.000,E1 32.752} C_DIS
LIN {X 0.086,Y -220.569,Z 510.165,A 0.000,B 0.000,C 90.000,E1 29.667} C_DIS
LIN {X -0.084,Y -214.699,Z 510.148,A 0.000,B 0.000,C 90.000,E1 26.616} C_DIS
LIN {X -0.003,Y -209.715,Z 510.130,A 0.000,B 0.000,C 90.000,E1 23.462} C_DIS
LIN {X -0.017,Y -204.611,Z 510.108,A 0.000,B 0.000,C 90.000,E1 19.504} C_DIS
LIN {X 0.047,Y -200.500,Z 510.086,A 0.000,B 0.000,C 90.000,E1 15.481} C_DIS
LIN {X -0.048,Y -196.878,Z 510.059,A 0.000,B 0.000,C 90.000,E1 10.658} C_DIS
LIN {X -0.017,Y -194.290,Z 510.023,A 0.000,B 0.000,C 90.000,E1 4.131} C_DIS
LIN {X -0.019,Y -195.756,Z 509.961,A 0.000,B 0.000,C 90.000,E1 352.996} C_DIS
LIN {X -0.004,Y -199.355,Z 509.929,A 0.000,B 0.000,C 90.000,E1 347.297} C_DIS
LIN {X -0.030,Y -203.138,Z 509.907,A 0.000,B 0.000,C 90.000,E1 343.268} C_DIS
LIN {X -0.020,Y -207.755,Z 509.885,A 0.000,B 0.000,C 90.000,E1 339.263} C_DIS
LIN {X 0.058,Y -213.135,Z 509.863,A 0.000,B 0.000,C 90.000,E1 335.281} C_DIS
LIN {X -0.011,Y -219.085,Z 509.841,A 0.000,B 0.000,C 90.000,E1 331.385} C_DIS
LIN {X -0.060,Y -225.647,Z 509.820,A 0.000,B 0.000,C 90.000,E1 327.533} C_DIS
LIN {X 0.020,Y -232.922,Z 509.798,A 0.000,B 0.000,C 90.000,E1 323.703} C_DIS
LIN {X -0.143,Y -240.718,Z 509.778,A 0.000,B 0.000,C 90.000,E1 319.989} C_DIS
LIN {X -0.148,Y -249.548,Z 509.757,A 0.000,B 0.000,C 90.000,E1 316.296} C_DIS
LIN {X -0.070,Y -258.590,Z 509.739,A 0.000,B 0.000,C 90.000,E1 313.014} C_DIS
LIN {X 0.029,Y -269.675,Z 509.719,A 0.000,B 0.000,C 90.000,E1 309.439} C_DIS
LIN {X 0.023,Y -282.122,Z 509.700,A 0.000,B 0.000,C 90.000,E1 305.964} C_DIS
LIN {X 0.152,Y -295.814,Z 509.681,A 0.000,B 0.000,C 90.000,E1 302.546} C_DIS
LIN {X -0.084,Y -310.467,Z 509.663,A 0.000,B 0.000,C 90.000,E1 299.283} C_DIS
LIN {X -0.053,Y -323.264,Z 509.648,A 0.000,B 0.000,C 90.000,E1 296.693} C_DIS
LIN {X 0.077,Y -333.898,Z 509.638,A 0.000,B 0.000,C 90.000,E1 294.771} C_DIS
LIN {X -0.167,Y -349.480,Z 509.624,A 0.000,B 0.000,C 90.000,E1 292.333} C_DIS
LIN {X 0.121,Y -368.990,Z 509.609,A 0.000,B 0.000,C 90.000,E1 289.577} C_DIS
LIN {X -0.109,Y -387.983,Z 509.596,A 0.000,B 0.000,C 90.000,E1 287.275} C_DIS
LIN {X -0.215,Y -412.715,Z 509.580,A 0.000,B 0.000,C 90.000,E1 284.481} C_DIS
LIN {X -0.164,Y -425.156,Z 509.573,A 0.000,B 0.000,C 90.000,E1 283.119} C_DIS
LIN {X -0.158,Y -437.311,Z 509.565,A 0.000,B 0.000,C 90.000,E1 281.771} C_DIS
LIN {X 0.241,Y -446.663,Z 509.559,A 0.000,B 0.000,C 90.000,E1 280.658} C_DIS
LIN {X -0.213,Y -455.339,Z 509.554,A 0.000,B 0.000,C 90.000,E1 279.670} C_DIS
LIN {X 0.059,Y -461.301,Z 509.549,A 0.000,B 0.000,C 90.000,E1 278.859} C_DIS
LIN {X -0.075,Y -466.657,Z 509.545,A 0.000,B 0.000,C 90.000,E1 278.106} C_DIS
LIN {X -0.160,Y -471.479,Z 509.541,A 0.000,B 0.000,C 90.000,E1 277.352} C_DIS
LIN {X 0.206,Y -475.771,Z 509.537,A 0.000,B 0.000,C 90.000,E1 276.549} C_DIS
LIN {X 0.198,Y -479.526,Z 509.532,A 0.000,B 0.000,C 90.000,E1 275.796} C_DIS
LIN {X 0.171,Y -482.738,Z 509.528,A 0.000,B 0.000,C 90.000,E1 275.049} C_DIS
LIN {X -0.140,Y -484.496,Z 509.525,A 0.000,B 0.000,C 90.000,E1 274.588} C_DIS
LIN {X 0.001,Y -485.951,Z 509.523,A 0.000,B 0.000,C 90.000,E1 274.073} C_DIS
LIN {X 0.189,Y -487.005,Z 509.520,A 0.000,B 0.000,C 90.000,E1 273.555} C_DIS
LIN {X -0.106,Y -487.786,Z 509.517,A 0.000,B 0.000,C 90.000,E1 273.094} C_DIS
LIN {X 0.067,Y -488.216,Z 509.514,A 0.000,B 0.000,C 90.000,E1 272.579} C_DIS
LIN {X -0.241,Y -488.259,Z 509.512,A 0.000,B 0.000,C 90.000,E1 272.121} C_DIS
LIN {X -0.043,Y -487.911,Z 509.509,A 0.000,B 0.000,C 90.000,E1 271.604} C_DIS
LIN {X 0.140,Y -487.159,Z 509.506,A 0.000,B 0.000,C 90.000,E1 271.088} C_DIS
LIN {X -0.164,Y -485.974,Z 509.503,A 0.000,B 0.000,C 90.000,E1 270.630} C_DIS
LIN {X 0.014,Y -484.227,Z 509.501,A 0.000,B 0.000,C 90.000,E1 270.115} C_DIS
LIN {X 0.184,Y -481.823,Z 509.498,A 0.000,B 0.000,C 90.000,E1 269.599} C_DIS
LIN {X -0.144,Y -478.677,Z 509.495,A 0.000,B 0.000,C 90.000,E1 269.141} C_DIS
LIN {X -0.008,Y -474.683,Z 509.492,A 0.000,B 0.000,C 90.000,E1 268.625} C_DIS
LIN {X 0.119,Y -469.620,Z 509.490,A 0.000,B 0.000,C 90.000,E1 268.108} C_DIS
LIN {X -0.047,Y -463.552,Z 509.487,A 0.000,B 0.000,C 90.000,E1 267.650} C_DIS
LIN {X 0.147,Y -460.417,Z 509.486,A 0.000,B 0.000,C 90.000,E1 267.421} C_DIS
LIN {X -0.071,Y -453.664,Z 509.484,A 0.000,B 0.000,C 90.000,E1 267.078} C_DIS
LIN {X -0.207,Y -446.844,Z 509.482,A 0.000,B 0.000,C 90.000,E1 266.788} C_DIS
LIN {X -0.016,Y -439.819,Z 509.481,A 0.000,B 0.000,C 90.000,E1 266.502} C_DIS
LIN {X 0.071,Y -432.376,Z 509.479,A 0.000,B 0.000,C 90.000,E1 266.274} C_DIS
LIN {X 0.107,Y -423.698,Z 509.478,A 0.000,B 0.000,C 90.000,E1 266.102} C_DIS
LIN {X 0.014,Y -418.125,Z 509.478,A 0.000,B 0.000,C 90.000,E1 266.045} C_DIS
LIN {X 0.026,Y -409.563,Z 509.478,A 0.000,B 0.000,C 90.000,E1 265.988} C_DIS
LIN {X -0.023,Y -180.919,Z 509.478,A 0.000,B 0.000,C 90.000,E1 265.988} C_DIS
LIN {X -0.022,Y -180.884,Z 509.473,A 0.000,B 0.000,C 90.000,E1 265.122} C_DIS
LIN {X 0.037,Y -179.005,Z 509.445,A 0.000,B 0.000,C 90.000,E1 260.038} C_DIS
LIN {X -0.044,Y -178.609,Z 509.440,A 0.000,B 0.000,C 90.000,E1 259.218} C_DIS
LIN {X 0.024,Y -175.662,Z 509.412,A 0.000,B 0.000,C 90.000,E1 254.102} C_DIS
LIN {X 0.029,Y -172.379,Z 509.388,A 0.000,B 0.000,C 90.000,E1 249.826} C_DIS
LIN {X 0.043,Y -171.177,Z 509.378,A 0.000,B 0.000,C 90.000,E1 248.103} C_DIS
LIN {X 0.087,Y -167.471,Z 509.354,A 0.000,B 0.000,C 90.000,E1 243.768} C_DIS
LIN {X 0.020,Y -166.868,Z 509.350,A 0.000,B 0.000,C 90.000,E1 242.922} C_DIS
LIN {X 0.074,Y -162.172,Z 509.320,A 0.000,B 0.000,C 90.000,E1 237.661} C_DIS
LIN {X -0.005,Y -160.736,Z 509.311,A 0.000,B 0.000,C 90.000,E1 235.928} C_DIS
LIN {X -0.026,Y -157.538,Z 509.291,A 0.000,B 0.000,C 90.000,E1 232.396} C_DIS
LIN {X 0.031,Y -155.564,Z 509.276,A 0.000,B 0.000,C 90.000,E1 229.703} C_DIS
LIN {X -0.036,Y -151.853,Z 509.251,A 0.000,B 0.000,C 90.000,E1 225.243} C_DIS
LIN {X -0.021,Y -150.074,Z 509.236,A 0.000,B 0.000,C 90.000,E1 222.528} C_DIS
LIN {X 0.013,Y -146.880,Z 509.211,A 0.000,B 0.000,C 90.000,E1 217.971} C_DIS
LIN {X 0.002,Y -145.466,Z 509.196,A 0.000,B 0.000,C 90.000,E1 215.231} C_DIS
LIN {X -0.081,Y -142.879,Z 509.170,A 0.000,B 0.000,C 90.000,E1 210.669} C_DIS
LIN {X -0.024,Y -141.497,Z 509.150,A 0.000,B 0.000,C 90.000,E1 206.950} C_DIS
LIN {X 0.025,Y -139.387,Z 509.114,A 0.000,B 0.000,C 90.000,E1 200.429} C_DIS
LIN {X 0.013,Y -138.844,Z 509.098,A 0.000,B 0.000,C 90.000,E1 197.638} C_DIS
LIN {X -0.063,Y -138.353,Z 509.057,A 0.000,B 0.000,C 90.000,E1 190.197} C_DIS
LIN {X 0.069,Y -139.518,Z 509.005,A 0.000,B 0.000,C 90.000,E1 180.802} C_DIS
LIN {X 0.010,Y -141.176,Z 508.974,A 0.000,B 0.000,C 90.000,E1 175.241} C_DIS
LIN {X -0.018,Y -142.555,Z 508.958,A 0.000,B 0.000,C 90.000,E1 172.470} C_DIS
LIN {X 0.049,Y -144.833,Z 508.932,A 0.000,B 0.000,C 90.000,E1 167.825} C_DIS
LIN {X 0.034,Y -147.456,Z 508.912,A 0.000,B 0.000,C 90.000,E1 164.157} C_DIS
LIN {X -0.079,Y -150.038,Z 508.892,A 0.000,B 0.000,C 90.000,E1 160.550} C_DIS
LIN {X -0.073,Y -153.379,Z 508.872,A 0.000,B 0.000,C 90.000,E1 156.922} C_DIS
LIN {X -0.026,Y -155.911,Z 508.857,A 0.000,B 0.000,C 90.000,E1 154.204} C_DIS
LIN {X 0.089,Y -159.774,Z 508.837,A 0.000,B 0.000,C 90.000,E1 150.589} C_DIS
LIN {X -0.063,Y -162.014,Z 508.827,A 0.000,B 0.000,C 90.000,E1 148.869} C_DIS
LIN {X 0.050,Y -166.207,Z 508.807,A 0.000,B 0.000,C 90.000,E1 145.308} C_DIS
LIN {X 0.053,Y -171.223,Z 508.788,A 0.000,B 0.000,C 90.000,E1 141.823} C_DIS
LIN {X -0.024,Y -176.110,Z 508.769,A 0.000,B 0.000,C 90.000,E1 138.405} C_DIS
LIN {X 0.093,Y -180.373,Z 508.755,A 0.000,B 0.000,C 90.000,E1 135.810} C_DIS
LIN {X 0.070,Y -185.781,Z 508.736,A 0.000,B 0.000,C 90.000,E1 132.447} C_DIS
LIN {X 0.003,Y -190.397,Z 508.722,A 0.000,B 0.000,C 90.000,E1 129.967} C_DIS
LIN {X 0.070,Y -192.556,Z 508.715,A 0.000,B 0.000,C 90.000,E1 128.669} C_DIS
LIN {X 0.070,Y -289.226,Z 508.715,A 0.000,B 0.000,C 90.000,E1 128.669} C_DIS
LIN {X 0.035,Y -290.087,Z 508.715,A 0.000,B 0.000,C 90.000,E1 128.669} C_DIS
LIN {X 0.168,Y -295.012,Z 508.714,A 0.000,B 0.000,C 90.000,E1 128.463} C_DIS
LIN {X 0.069,Y -297.401,Z 508.713,A 0.000,B 0.000,C 90.000,E1 128.302} C_DIS
LIN {X -0.129,Y -301.248,Z 508.710,A 0.000,B 0.000,C 90.000,E1 127.890} C_DIS
LIN {X 0.123,Y -303.139,Z 508.709,A 0.000,B 0.000,C 90.000,E1 127.523} C_DIS
LIN {X -0.051,Y -304.624,Z 508.707,A 0.000,B 0.000,C 90.000,E1 127.237} C_DIS
LIN {X 0.151,Y -305.836,Z 508.705,A 0.000,B 0.000,C 90.000,E1 126.870} C_DIS
LIN {X 0.123,Y -316.803,Z 508.685,A 0.000,B 0.000,C 90.000,E1 123.293} C_DIS
LIN {X -0.133,Y -327.120,Z 508.669,A 0.000,B 0.000,C 90.000,E1 120.463} C_DIS
LIN {X -0.151,Y -338.793,Z 508.653,A 0.000,B 0.000,C 90.000,E1 117.641} C_DIS
LIN {X 0.014,Y -351.919,Z 508.638,A 0.000,B 0.000,C 90.000,E1 114.847} C_DIS
LIN {X -0.122,Y -364.907,Z 508.625,A 0.000,B 0.000,C 90.000,E1 112.461} C_DIS
LIN {X 0.130,Y -379.233,Z 508.612,A 0.000,B 0.000,C 90.000,E1 110.066} C_DIS
LIN {X 0.137,Y -395.003,Z 508.599,A 0.000,B 0.000,C 90.000,E1 107.764} C_DIS
LIN {X -0.089,Y -412.331,Z 508.586,A 0.000,B 0.000,C 90.000,E1 105.552} C_DIS
LIN {X -0.002,Y -431.335,Z 508.574,A 0.000,B 0.000,C 90.000,E1 103.355} C_DIS
LIN {X 0.020,Y -451.451,Z 508.563,A 0.000,B 0.000,C 90.000,E1 101.299} C_DIS
LIN {X -0.128,Y -472.113,Z 508.552,A 0.000,B 0.000,C 90.000,E1 99.434} C_DIS
LIN {X 0.049,Y -479.811,Z 508.549,A 0.000,B 0.000,C 90.000,E1 98.746} C_DIS
LIN {X 0.092,Y -481.747,Z 508.547,A 0.000,B 0.000,C 90.000,E1 98.511} C_DIS
LIN {X 0.136,Y -483.228,Z 508.546,A 0.000,B 0.000,C 90.000,E1 98.276} C_DIS
LIN {X -0.053,Y -484.446,Z 508.545,A 0.000,B 0.000,C 90.000,E1 98.049} C_DIS
LIN {X -0.173,Y -485.337,Z 508.543,A 0.000,B 0.000,C 90.000,E1 97.814} C_DIS
LIN {X 0.015,Y -486.288,Z 508.541,A 0.000,B 0.000,C 90.000,E1 97.296} C_DIS
LIN {X 0.210,Y -486.247,Z 508.538,A 0.000,B 0.000,C 90.000,E1 96.777} C_DIS
LIN {X -0.074,Y -485.207,Z 508.535,A 0.000,B 0.000,C 90.000,E1 96.315} C_DIS
LIN {X -0.240,Y -484.265,Z 508.534,A 0.000,B 0.000,C 90.000,E1 96.087} C_DIS
LIN {X 0.125,Y -482.982,Z 508.532,A 0.000,B 0.000,C 90.000,E1 95.796} C_DIS
LIN {X -0.045,Y -481.264,Z 508.531,A 0.000,B 0.000,C 90.000,E1 95.568} C_DIS
LIN {X 0.094,Y -461.354,Z 508.517,A 0.000,B 0.000,C 90.000,E1 93.037} C_DIS
LIN {X 0.141,Y -450.624,Z 508.508,A 0.000,B 0.000,C 90.000,E1 91.489} C_DIS
LIN {X -0.081,Y -437.638,Z 508.497,A 0.000,B 0.000,C 90.000,E1 89.427} C_DIS
LIN {X 0.146,Y -426.224,Z 508.486,A 0.000,B 0.000,C 90.000,E1 87.535} C_DIS
LIN {X -0.169,Y -413.355,Z 508.474,A 0.000,B 0.000,C 90.000,E1 85.412} C_DIS
LIN {X 0.103,Y -400.753,Z 508.462,A 0.000,B 0.000,C 90.000,E1 83.166} C_DIS
LIN {X 0.057,Y -391.416,Z 508.453,A 0.000,B 0.000,C 90.000,E1 81.489} C_DIS
LIN {X -0.059,Y -380.397,Z 508.442,A 0.000,B 0.000,C 90.000,E1 79.511} C_DIS
LIN {X 0.045,Y -369.436,Z 508.430,A 0.000,B 0.000,C 90.000,E1 77.465} C_DIS
LIN {X 0.043,Y -357.824,Z 508.417,A 0.000,B 0.000,C 90.000,E1 75.102} C_DIS
LIN {X -0.068,Y -348.629,Z 508.406,A 0.000,B 0.000,C 90.000,E1 73.015} C_DIS
LIN {X 0.067,Y -338.278,Z 508.390,A 0.000,B 0.000,C 90.000,E1 70.242} C_DIS
LIN {X -0.051,Y -327.806,Z 508.373,A 0.000,B 0.000,C 90.000,E1 67.155} C_DIS
LIN {X 0.185,Y -319.901,Z 508.359,A 0.000,B 0.000,C 90.000,E1 64.588} C_DIS
LIN {X 0.200,Y -312.075,Z 508.345,A 0.000,B 0.000,C 90.000,E1 62.025} C_DIS
LIN {X -0.043,Y -306.199,Z 508.334,A 0.000,B 0.000,C 90.000,E1 60.127} C_DIS
LIN {X -0.029,Y -298.444,Z 508.319,A 0.000,B 0.000,C 90.000,E1 57.502} C_DIS
LIN {X -0.143,Y -289.248,Z 508.301,A 0.000,B 0.000,C 90.000,E1 54.196} C_DIS
LIN {X -0.010,Y -283.999,Z 508.290,A 0.000,B 0.000,C 90.000,E1 52.145} C_DIS
LIN {X -0.073,Y -278.510,Z 508.278,A 0.000,B 0.000,C 90.000,E1 50.114} C_DIS
LIN {X -0.018,Y -274.619,Z 508.271,A 0.000,B 0.000,C 90.000,E1 48.728} C_DIS
LIN {X 0.026,Y -269.318,Z 508.261,A 0.000,B 0.000,C 90.000,E1 46.986} C_DIS
LIN {X 0.035,Y -262.427,Z 508.249,A 0.000,B 0.000,C 90.000,E1 44.879} C_DIS
LIN {X -0.039,Y -253.147,Z 508.234,A 0.000,B 0.000,C 90.000,E1 42.043} C_DIS
LIN {X 0.066,Y -243.188,Z 508.215,A 0.000,B 0.000,C 90.000,E1 38.749} C_DIS
LIN {X 0.020,Y -234.929,Z 508.199,A 0.000,B 0.000,C 90.000,E1 35.804} C_DIS
LIN {X 0.012,Y -227.350,Z 508.182,A 0.000,B 0.000,C 90.000,E1 32.801} C_DIS
LIN {X 0.027,Y -220.648,Z 508.165,A 0.000,B 0.000,C 90.000,E1 29.745} C_DIS
LIN {X -0.038,Y -214.760,Z 508.148,A 0.000,B 0.000,C 90.000,E1 26.668} C_DIS
LIN {X 0.038,Y -209.777,Z 508.131,A 0.000,B 0.000,C 90.000,E1 23.515} C_DIS
LIN {X -0.048,Y -204.656,Z 508.109,A 0.000,B 0.000,C 90.000,E1 19.577} C_DIS
LIN {X 0.026,Y -200.514,Z 508.086,A 0.000,B 0.000,C 90.000,E1 15.552} C_DIS
LIN {X -0.018,Y -196.866,Z 508.060,A 0.000,B 0.000,C 90.000,E1 10.715} C_DIS
LIN {X 0.008,Y -194.238,Z 508.023,A 0.000,B 0.000,C 90.000,E1 4.188} C_DIS
LIN {X -0.024,Y -195.638,Z 507.961,A 0.000,B 0.000,C 90.000,E1 352.996} C_DIS
LIN {X -0.015,Y -199.225,Z 507.929,A 0.000,B 0.000,C 90.000,E1 347.297} C_DIS
LIN {X -0.046,Y -202.999,Z 507.907,A 0.000,B 0.000,C 90.000,E1 343.268} C_DIS
LIN {X -0.041,Y -207.611,Z 507.885,A 0.000,B 0.000,C 90.000,E1 339.263} C_DIS
LIN {X 0.033,Y -212.994,Z 507.863,A 0.000,B 0.000,C 90.000,E1 335.281} C_DIS
LIN {X -0.041,Y -218.952,Z 507.841,A 0.000,B 0.000,C 90.000,E1 331.385} C_DIS
LIN {X 0.027,Y -225.534,Z 507.819,A 0.000,B 0.000,C 90.000,E1 327.502} C_DIS
LIN {X -0.021,Y -232.816,Z 507.798,A 0.000,B 0.000,C 90.000,E1 323.703} C_DIS
LIN {X 0.151,Y -240.638,Z 507.777,A 0.000,B 0.000,C 90.000,E1 319.908} C_DIS
LIN {X -0.006,Y -247.608,Z 507.761,A 0.000,B 0.000,C 90.000,E1 316.986} C_DIS
LIN {X 0.011,Y -256.422,Z 507.743,A 0.000,B 0.000,C 90.000,E1 313.704} C_DIS
LIN {X 0.009,Y -267.334,Z 507.723,A 0.000,B 0.000,C 90.000,E1 310.135} C_DIS
LIN {X -0.090,Y -279.519,Z 507.704,A 0.000,B 0.000,C 90.000,E1 306.664} C_DIS
LIN {X -0.051,Y -293.019,Z 507.685,A 0.000,B 0.000,C 90.000,E1 303.245} C_DIS
LIN {X -0.069,Y -307.428,Z 507.666,A 0.000,B 0.000,C 90.000,E1 299.922} C_DIS
LIN {X -0.055,Y -321.598,Z 507.650,A 0.000,B 0.000,C 90.000,E1 297.001} C_DIS
LIN {X 0.006,Y -333.922,Z 507.638,A 0.000,B 0.000,C 90.000,E1 294.771} C_DIS
LIN {X 0.084,Y -349.506,Z 507.624,A 0.000,B 0.000,C 90.000,E1 292.280} C_DIS
LIN {X 0.045,Y -369.034,Z 507.609,A 0.000,B 0.000,C 90.000,E1 289.577} C_DIS
LIN {X 0.181,Y -388.018,Z 507.596,A 0.000,B 0.000,C 90.000,E1 287.221} C_DIS
LIN {X -0.166,Y -412.613,Z 507.580,A 0.000,B 0.000,C 90.000,E1 284.481} C_DIS
LIN {X -0.039,Y -424.994,Z 507.573,A 0.000,B 0.000,C 90.000,E1 283.119} C_DIS
LIN {X 0.004,Y -437.157,Z 507.565,A 0.000,B 0.000,C 90.000,E1 281.771} C_DIS
LIN {X -0.035,Y -446.549,Z 507.560,A 0.000,B 0.000,C 90.000,E1 280.715} C_DIS
LIN {X -0.047,Y -455.287,Z 507.554,A 0.000,B 0.000,C 90.000,E1 279.670} C_DIS
LIN {X 0.226,Y -461.262,Z 507.549,A 0.000,B 0.000,C 90.000,E1 278.859} C_DIS
LIN {X 0.094,Y -466.640,Z 507.545,A 0.000,B 0.000,C 90.000,E1 278.106} C_DIS
LIN {X 0.010,Y -471.475,Z 507.541,A 0.000,B 0.000,C 90.000,E1 277.352} C_DIS
LIN {X -0.096,Y -475.804,Z 507.537,A 0.000,B 0.000,C 90.000,E1 276.606} C_DIS
LIN {X -0.105,Y -479.522,Z 507.532,A 0.000,B 0.000,C 90.000,E1 275.853} C_DIS
LIN {X 0.047,Y -481.745,Z 507.530,A 0.000,B 0.000,C 90.000,E1 275.334} C_DIS
LIN {X 0.035,Y -484.527,Z 507.526,A 0.000,B 0.000,C 90.000,E1 274.588} C_DIS
LIN {X 0.177,Y -485.975,Z 507.523,A 0.000,B 0.000,C 90.000,E1 274.073} C_DIS
LIN {X -0.121,Y -487.090,Z 507.520,A 0.000,B 0.000,C 90.000,E1 273.612} C_DIS
LIN {X 0.072,Y -487.863,Z 507.517,A 0.000,B 0.000,C 90.000,E1 273.094} C_DIS
LIN {X 0.244,Y -488.331,Z 507.514,A 0.000,B 0.000,C 90.000,E1 272.579} C_DIS
LIN {X -0.064,Y -488.393,Z 507.512,A 0.000,B 0.000,C 90.000,E1 272.121} C_DIS
LIN {X 0.136,Y -488.063,Z 507.509,A 0.000,B 0.000,C 90.000,E1 271.604} C_DIS
LIN {X -0.169,Y -487.343,Z 507.506,A 0.000,B 0.000,C 90.000,E1 271.146} C_DIS
LIN {X 0.014,Y -486.132,Z 507.504,A 0.000,B 0.000,C 90.000,E1 270.630} C_DIS
LIN {X 0.193,Y -484.409,Z 507.501,A 0.000,B 0.000,C 90.000,E1 270.115} C_DIS
LIN {X -0.119,Y -482.026,Z 507.498,A 0.000,B 0.000,C 90.000,E1 269.656} C_DIS
LIN {X 0.035,Y -478.937,Z 507.495,A 0.000,B 0.000,C 90.000,E1 269.141} C_DIS
LIN {X 0.171,Y -474.943,Z 507.492,A 0.000,B 0.000,C 90.000,E1 268.625} C_DIS
LIN {X -0.172,Y -469.926,Z 507.490,A 0.000,B 0.000,C 90.000,E1 268.165} C_DIS
LIN {X 0.217,Y -467.122,Z 507.488,A 0.000,B 0.000,C 90.000,E1 267.879} C_DIS
LIN {X -0.126,Y -460.894,Z 507.486,A 0.000,B 0.000,C 90.000,E1 267.478} C_DIS
LIN {X 0.093,Y -454.174,Z 507.484,A 0.000,B 0.000,C 90.000,E1 267.078} C_DIS
LIN {X -0.083,Y -447.393,Z 507.482,A 0.000,B 0.000,C 90.000,E1 266.788} C_DIS
LIN {X 0.100,Y -440.483,Z 507.481,A 0.000,B 0.000,C 90.000,E1 266.502} C_DIS
LIN {X 0.202,Y -433.192,Z 507.479,A 0.000,B 0.000,C 90.000,E1 266.274} C_DIS
LIN {X -0.206,Y -424.940,Z 507.479,A 0.000,B 0.000,C 90.000,E1 266.159} C_DIS
LIN {X 0.178,Y -414.036,Z 507.478,A 0.000,B 0.000,C 90.000,E1 265.988} C_DIS
LIN {X 0.013,Y -409.889,Z 507.478,A 0.000,B 0.000,C 90.000,E1 265.988} C_DIS
LIN {X -0.030,Y -180.920,Z 507.478,A 0.000,B 0.000,C 90.000,E1 265.988} C_DIS
LIN {X 0.010,Y -180.851,Z 507.472,A 0.000,B 0.000,C 90.000,E1 264.951} C_DIS
LIN {X 0.086,Y -178.899,Z 507.443,A 0.000,B 0.000,C 90.000,E1 259.690} C_DIS
LIN {X -0.010,Y -175.942,Z 507.415,A 0.000,B 0.000,C 90.000,E1 254.629} C_DIS
LIN {X -0.063,Y -175.398,Z 507.410,A 0.000,B 0.000,C 90.000,E1 253.795} C_DIS
LIN {X -0.058,Y -172.167,Z 507.386,A 0.000,B 0.000,C 90.000,E1 249.518} C_DIS
LIN {X -0.020,Y -171.636,Z 507.381,A 0.000,B 0.000,C 90.000,E1 248.646} C_DIS
LIN {X -0.024,Y -167.858,Z 507.357,A 0.000,B 0.000,C 90.000,E1 244.332} C_DIS
LIN {X -0.081,Y -166.590,Z 507.348,A 0.000,B 0.000,C 90.000,E1 242.615} C_DIS
LIN {X 0.052,Y -162.581,Z 507.323,A 0.000,B 0.000,C 90.000,E1 238.201} C_DIS
LIN {X 0.022,Y -161.263,Z 507.314,A 0.000,B 0.000,C 90.000,E1 236.453} C_DIS
LIN {X 0.021,Y -157.264,Z 507.289,A 0.000,B 0.000,C 90.000,E1 232.029} C_DIS
LIN {X -0.052,Y -155.985,Z 507.279,A 0.000,B 0.000,C 90.000,E1 230.275} C_DIS
LIN {X -0.091,Y -152.241,Z 507.254,A 0.000,B 0.000,C 90.000,E1 225.810} C_DIS
LIN {X 0.034,Y -150.481,Z 507.239,A 0.000,B 0.000,C 90.000,E1 223.056} C_DIS
LIN {X -0.038,Y -147.206,Z 507.214,A 0.000,B 0.000,C 90.000,E1 218.543} C_DIS
LIN {X -0.067,Y -145.227,Z 507.194,A 0.000,B 0.000,C 90.000,E1 214.898} C_DIS
LIN {X 0.044,Y -142.353,Z 507.163,A 0.000,B 0.000,C 90.000,E1 209.333} C_DIS
LIN {X -0.029,Y -141.740,Z 507.153,A 0.000,B 0.000,C 90.000,E1 207.513} C_DIS
LIN {X 0.077,Y -139.488,Z 507.117,A 0.000,B 0.000,C 90.000,E1 200.972} C_DIS
LIN {X 0.066,Y -138.990,Z 507.101,A 0.000,B 0.000,C 90.000,E1 198.181} C_DIS
LIN {X 0.027,Y -138.335,Z 507.054,A 0.000,B 0.000,C 90.000,E1 189.792} C_DIS
LIN {X 0.052,Y -139.419,Z 507.008,A 0.000,B 0.000,C 90.000,E1 181.375} C_DIS
LIN {X -0.035,Y -141.339,Z 506.972,A 0.000,B 0.000,C 90.000,E1 174.894} C_DIS
LIN {X -0.078,Y -142.695,Z 506.956,A 0.000,B 0.000,C 90.000,E1 172.129} C_DIS
LIN {X 0.043,Y -145.060,Z 506.930,A 0.000,B 0.000,C 90.000,E1 167.465} C_DIS
LIN {X 0.040,Y -147.686,Z 506.910,A 0.000,B 0.000,C 90.000,E1 163.795} C_DIS
LIN {X -0.068,Y -150.333,Z 506.890,A 0.000,B 0.000,C 90.000,E1 160.188} C_DIS
LIN {X 0.003,Y -153.750,Z 506.870,A 0.000,B 0.000,C 90.000,E1 156.538} C_DIS
LIN {X -0.005,Y -157.164,Z 506.850,A 0.000,B 0.000,C 90.000,E1 152.948} C_DIS
LIN {X -0.072,Y -161.317,Z 506.830,A 0.000,B 0.000,C 90.000,E1 149.410} C_DIS
LIN {X 0.082,Y -164.431,Z 506.815,A 0.000,B 0.000,C 90.000,E1 146.707} C_DIS
LIN {X 0.076,Y -169.117,Z 506.796,A 0.000,B 0.000,C 90.000,E1 143.210} C_DIS
LIN {X 0.025,Y -171.671,Z 506.786,A 0.000,B 0.000,C 90.000,E1 141.492} C_DIS
LIN {X -0.064,Y -176.638,Z 506.767,A 0.000,B 0.000,C 90.000,E1 138.081} C_DIS
LIN {X 0.063,Y -180.935,Z 506.753,A 0.000,B 0.000,C 90.000,E1 135.486} C_DIS
LIN {X 0.052,Y -186.355,Z 506.734,A 0.000,B 0.000,C 90.000,E1 132.123} C_DIS
LIN {X -0.008,Y -190.987,Z 506.720,A 0.000,B 0.000,C 90.000,E1 129.644} C_DIS
LIN {X -0.053,Y -192.618,Z 506.715,A 0.000,B 0.000,C 90.000,E1 128.669} C_DIS
LIN {X -0.115,Y -289.857,Z 506.715,A 0.000,B 0.000,C 90.000,E1 128.669} C_DIS
LIN {X -0.093,Y -291.936,Z 506.714,A 0.000,B 0.000,C 90.000,E1 128.624} C_DIS
LIN {X -0.019,Y -297.286,Z 506.713,A 0.000,B 0.000,C 90.000,E1 128.302} C_DIS
LIN {X -0.128,Y -300.165,Z 506.711,A 0.000,B 0.000,C 90.000,E1 128.016} C_DIS
LIN {X 0.048,Y -302.203,Z 506.709,A 0.000,B 0.000,C 90.000,E1 127.684} C_DIS
LIN {X -0.015,Y -303.803,Z 506.708,A 0.000,B 0.000,C 90.000,E1 127.397} C_DIS
LIN {X -0.060,Y -305.205,Z 506.706,A 0.000,B 0.000,C 90.000,E1 127.076} C_DIS
LIN {X -0.045,Y -306.311,Z 506.704,A 0.000,B 0.000,C 90.000,E1 126.744} C_DIS
LIN {X -0.122,Y -316.244,Z 506.686,A 0.000,B 0.000,C 90.000,E1 123.499} C_DIS
LIN {X 0.046,Y -326.489,Z 506.670,A 0.000,B 0.000,C 90.000,E1 120.590} C_DIS
LIN {X 0.013,Y -338.083,Z 506.654,A 0.000,B 0.000,C 90.000,E1 117.769} C_DIS
LIN {X -0.154,Y -351.124,Z 506.639,A 0.000,B 0.000,C 90.000,E1 115.027} C_DIS
LIN {X 0.014,Y -364.031,Z 506.626,A 0.000,B 0.000,C 90.000,E1 112.589} C_DIS
LIN {X -0.104,Y -378.270,Z 506.612,A 0.000,B 0.000,C 90.000,E1 110.248} C_DIS
LIN {X -0.130,Y -393.946,Z 506.600,A 0.000,B 0.000,C 90.000,E1 107.946} C_DIS
LIN {X 0.113,Y -411.173,Z 506.587,A 0.000,B 0.000,C 90.000,E1 105.662} C_DIS
LIN {X 0.065,Y -430.077,Z 506.575,A 0.000,B 0.000,C 90.000,E1 103.480} C_DIS
LIN {X 0.011,Y -450.155,Z 506.563,A 0.000,B 0.000,C 90.000,E1 101.422} C_DIS
LIN {X -0.212,Y -470.786,Z 506.553,A 0.000,B 0.000,C 90.000,E1 99.557} C_DIS
LIN {X 0.009,Y -478.659,Z 506.549,A 0.000,B 0.000,C 90.000,E1 98.859} C_DIS
LIN {X 0.134,Y -480.848,Z 506.548,A 0.000,B 0.000,C 90.000,E1 98.624} C_DIS
LIN {X 0.188,Y -482.516,Z 506.547,A 0.000,B 0.000,C 90.000,E1 98.398} C_DIS
LIN {X 0.067,Y -483.959,Z 506.545,A 0.000,B 0.000,C 90.000,E1 98.163} C_DIS
LIN {X -0.124,Y -485.035,Z 506.544,A 0.000,B 0.000,C 90.000,E1 97.936} C_DIS
LIN {X 0.127,Y -486.294,Z 506.541,A 0.000,B 0.000,C 90.000,E1 97.409} C_DIS
LIN {X -0.163,Y -486.534,Z 506.538,A 0.000,B 0.000,C 90.000,E1 96.947} C_DIS
LIN {X 0.035,Y -485.792,Z 506.536,A 0.000,B 0.000,C 90.000,E1 96.429} C_DIS
LIN {X 0.235,Y -483.942,Z 506.533,A 0.000,B 0.000,C 90.000,E1 95.910} C_DIS
LIN {X 0.068,Y -482.491,Z 506.532,A 0.000,B 0.000,C 90.000,E1 95.682} C_DIS
LIN {X -0.061,Y -474.512,Z 506.526,A 0.000,B 0.000,C 90.000,E1 94.702} C_DIS
LIN {X 0.030,Y -460.711,Z 506.516,A 0.000,B 0.000,C 90.000,E1 92.922} C_DIS
LIN {X 0.067,Y -450.049,Z 506.508,A 0.000,B 0.000,C 90.000,E1 91.375} C_DIS
LIN {X -0.165,Y -437.048,Z 506.496,A 0.000,B 0.000,C 90.000,E1 89.312} C_DIS
LIN {X 0.047,Y -425.624,Z 506.486,A 0.000,B 0.000,C 90.000,E1 87.421} C_DIS
LIN {X 0.131,Y -412.757,Z 506.474,A 0.000,B 0.000,C 90.000,E1 85.241} C_DIS
LIN {X -0.021,Y -400.169,Z 506.461,A 0.000,B 0.000,C 90.000,E1 83.053} C_DIS
LIN {X -0.079,Y -390.807,Z 506.452,A 0.000,B 0.000,C 90.000,E1 81.376} C_DIS
LIN {X 0.171,Y -379.804,Z 506.441,A 0.000,B 0.000,C 90.000,E1 79.342} C_DIS
LIN {X -0.053,Y -365.827,Z 506.426,A 0.000,B 0.000,C 90.000,E1 76.756} C_DIS
LIN {X -0.188,Y -353.238,Z 506.411,A 0.000,B 0.000,C 90.000,E1 74.102} C_DIS
LIN {X 0.035,Y -344.584,Z 506.400,A 0.000,B 0.000,C 90.000,E1 71.945} C_DIS
LIN {X -0.169,Y -332.511,Z 506.381,A 0.000,B 0.000,C 90.000,E1 68.592} C_DIS
LIN {X 0.100,Y -322.401,Z 506.363,A 0.000,B 0.000,C 90.000,E1 65.409} C_DIS
LIN {X 0.039,Y -314.520,Z 506.349,A 0.000,B 0.000,C 90.000,E1 62.871} C_DIS
LIN {X 0.111,Y -308.678,Z 506.339,A 0.000,B 0.000,C 90.000,E1 60.923} C_DIS
LIN {X 0.022,Y -300.833,Z 506.324,A 0.000,B 0.000,C 90.000,E1 58.329} C_DIS
LIN {X -0.021,Y -291.443,Z 506.306,A 0.000,B 0.000,C 90.000,E1 55.022} C_DIS
LIN {X 0.044,Y -284.395,Z 506.291,A 0.000,B 0.000,C 90.000,E1 52.316} C_DIS
LIN {X 0.035,Y -278.950,Z 506.279,A 0.000,B 0.000,C 90.000,E1 50.275} C_DIS
LIN {X -0.116,Y -273.014,Z 506.268,A 0.000,B 0.000,C 90.000,E1 48.243} C_DIS
LIN {X 0.104,Y -267.557,Z 506.258,A 0.000,B 0.000,C 90.000,E1 46.458} C_DIS
LIN {X -0.064,Y -259.502,Z 506.245,A 0.000,B 0.000,C 90.000,E1 44.028} C_DIS
LIN {X 0.002,Y -249.178,Z 506.227,A 0.000,B 0.000,C 90.000,E1 40.782} C_DIS
LIN {X 0.024,Y -241.577,Z 506.212,A 0.000,B 0.000,C 90.000,E1 38.222} C_DIS
LIN {X 0.125,Y -233.452,Z 506.196,A 0.000,B 0.000,C 90.000,E1 35.231} C_DIS
LIN {X -0.049,Y -225.996,Z 506.179,A 0.000,B 0.000,C 90.000,E1 32.260} C_DIS
LIN {X -0.066,Y -219.466,Z 506.162,A 0.000,B 0.000,C 90.000,E1 29.205} C_DIS
LIN {X -0.069,Y -213.730,Z 506.145,A 0.000,B 0.000,C 90.000,E1 26.104} C_DIS
LIN {X -0.016,Y -208.939,Z 506.127,A 0.000,B 0.000,C 90.000,E1 22.950} C_DIS
LIN {X 0.062,Y -203.966,Z 506.105,A 0.000,B 0.000,C 90.000,E1 18.960} C_DIS
LIN {X 0.050,Y -199.952,Z 506.083,A 0.000,B 0.000,C 90.000,E1 14.954} C_DIS
LIN {X -0.099,Y -196.461,Z 506.056,A 0.000,B 0.000,C 90.000,E1 10.141} C_DIS
LIN {X 0.065,Y -193.922,Z 506.015,A 0.000,B 0.000,C 90.000,E1 2.751} C_DIS
LIN {X -0.030,Y -195.514,Z 505.961,A 0.000,B 0.000,C 90.000,E1 352.996} C_DIS
LIN {X -0.057,Y -198.483,Z 505.934,A 0.000,B 0.000,C 90.000,E1 348.117} C_DIS
LIN {X 0.032,Y -202.013,Z 505.911,A 0.000,B 0.000,C 90.000,E1 344.047} C_DIS
LIN {X -0.062,Y -206.467,Z 505.889,A 0.000,B 0.000,C 90.000,E1 340.061} C_DIS
LIN {X 0.083,Y -211.719,Z 505.867,A 0.000,B 0.000,C 90.000,E1 336.049} C_DIS
LIN {X -0.030,Y -217.576,Z 505.845,A 0.000,B 0.000,C 90.000,E1 332.153} C_DIS
LIN {X -0.043,Y -224.041,Z 505.824,A 0.000,B 0.000,C 90.000,E1 328.280} C_DIS
LIN {X -0.148,Y -231.210,Z 505.802,A 0.000,B 0.000,C 90.000,E1 324.482} C_DIS
LIN {X 0.005,Y -238.905,Z 505.782,A 0.000,B 0.000,C 90.000,E1 320.678} C_DIS
LIN {X -0.057,Y -247.528,Z 505.761,A 0.000,B 0.000,C 90.000,E1 316.986} C_DIS
LIN {X -0.043,Y -256.367,Z 505.743,A 0.000,B 0.000,C 90.000,E1 313.704} C_DIS
LIN {X 0.155,Y -267.301,Z 505.723,A 0.000,B 0.000,C 90.000,E1 310.092} C_DIS
LIN {X -0.150,Y -279.515,Z 505.704,A 0.000,B 0.000,C 90.000,E1 306.664} C_DIS
LIN {X 0.046,Y -293.022,Z 505.685,A 0.000,B 0.000,C 90.000,E1 303.214} C_DIS
LIN {X 0.099,Y -305.957,Z 505.668,A 0.000,B 0.000,C 90.000,E1 300.207} C_DIS
LIN {X -0.124,Y -321.609,Z 505.650,A 0.000,B 0.000,C 90.000,E1 297.001} C_DIS
LIN {X -0.065,Y -333.954,Z 505.638,A 0.000,B 0.000,C 90.000,E1 294.771} C_DIS
LIN {X 0.010,Y -349.534,Z 505.624,A 0.000,B 0.000,C 90.000,E1 292.280} C_DIS
LIN {X -0.102,Y -366.783,Z 505.610,A 0.000,B 0.000,C 90.000,E1 289.885} C_DIS
LIN {X 0.101,Y -388.060,Z 505.596,A 0.000,B 0.000,C 90.000,E1 287.221} C_DIS
LIN {X -0.101,Y -412.487,Z 505.580,A 0.000,B 0.000,C 90.000,E1 284.481} C_DIS
LIN {X -0.025,Y -424.970,Z 505.573,A 0.000,B 0.000,C 90.000,E1 283.119} C_DIS
LIN {X 0.013,Y -437.185,Z 505.565,A 0.000,B 0.000,C 90.000,E1 281.771} C_DIS
LIN {X -0.025,Y -446.607,Z 505.560,A 0.000,B 0.000,C 90.000,E1 280.715} C_DIS
LIN {X -0.036,Y -455.386,Z 505.554,A 0.000,B 0.000,C 90.000,E1 279.670} C_DIS
LIN {X -0.218,Y -461.360,Z 505.549,A 0.000,B 0.000,C 90.000,E1 278.916} C_DIS
LIN {X -0.057,Y -468.420,Z 505.544,A 0.000,B 0.000,C 90.000,E1 277.871} C_DIS
LIN {X -0.194,Y -473.123,Z 505.539,A 0.000,B 0.000,C 90.000,E1 277.125} C_DIS
LIN {X -0.226,Y -477.246,Z 505.535,A 0.000,B 0.000,C 90.000,E1 276.372} C_DIS
LIN {X 0.199,Y -480.819,Z 505.531,A 0.000,B 0.000,C 90.000,E1 275.568} C_DIS
LIN {X -0.119,Y -482.854,Z 505.528,A 0.000,B 0.000,C 90.000,E1 275.106} C_DIS
LIN {X 0.047,Y -484.634,Z 505.526,A 0.000,B 0.000,C 90.000,E1 274.588} C_DIS
LIN {X 0.190,Y -486.060,Z 505.523,A 0.000,B 0.000,C 90.000,E1 274.073} C_DIS
LIN {X -0.108,Y -487.197,Z 505.520,A 0.000,B 0.000,C 90.000,E1 273.612} C_DIS
LIN {X 0.085,Y -487.974,Z 505.517,A 0.000,B 0.000,C 90.000,E1 273.094} C_DIS
LIN {X -0.229,Y -488.446,Z 505.514,A 0.000,B 0.000,C 90.000,E1 272.636} C_DIS
LIN {X -0.049,Y -488.521,Z 505.512,A 0.000,B 0.000,C 90.000,E1 272.121} C_DIS
LIN {X 0.151,Y -488.220,Z 505.509,A 0.000,B 0.000,C 90.000,E1 271.604} C_DIS
LIN {X -0.153,Y -487.494,Z 505.506,A 0.000,B 0.000,C 90.000,E1 271.146} C_DIS
LIN {X 0.032,Y -486.252,Z 505.504,A 0.000,B 0.000,C 90.000,E1 270.630} C_DIS
LIN {X 0.211,Y -484.515,Z 505.501,A 0.000,B 0.000,C 90.000,E1 270.115} C_DIS
LIN {X -0.100,Y -482.146,Z 505.498,A 0.000,B 0.000,C 90.000,E1 269.656} C_DIS
LIN {X 0.218,Y -480.727,Z 505.497,A 0.000,B 0.000,C 90.000,E1 269.370} C_DIS
LIN {X -0.115,Y -477.187,Z 505.494,A 0.000,B 0.000,C 90.000,E1 268.912} C_DIS
LIN {X 0.191,Y -475.094,Z 505.492,A 0.000,B 0.000,C 90.000,E1 268.625} C_DIS
LIN {X -0.152,Y -470.084,Z 505.490,A 0.000,B 0.000,C 90.000,E1 268.165} C_DIS
LIN {X 0.122,Y -463.984,Z 505.487,A 0.000,B 0.000,C 90.000,E1 267.650} C_DIS
LIN {X 0.045,Y -457.412,Z 505.485,A 0.000,B 0.000,C 90.000,E1 267.249} C_DIS
LIN {X 0.054,Y -450.624,Z 505.483,A 0.000,B 0.000,C 90.000,E1 266.906} C_DIS
LIN {X 0.050,Y -443.579,Z 505.481,A 0.000,B 0.000,C 90.000,E1 266.617} C_DIS
LIN {X -0.005,Y -436.556,Z 505.480,A 0.000,B 0.000,C 90.000,E1 266.388} C_DIS
LIN {X -0.169,Y -428.656,Z 505.479,A 0.000,B 0.000,C 90.000,E1 266.216} C_DIS
LIN {X 0.051,Y -419.055,Z 505.478,A 0.000,B 0.000,C 90.000,E1 266.045} C_DIS
LIN {X -0.026,Y -408.021,Z 505.478,A 0.000,B 0.000,C 90.000,E1 265.988} C_DIS
LIN {X -0.047,Y -180.919,Z 505.478,A 0.000,B 0.000,C 90.000,E1 265.988} C_DIS
LIN {X -0.006,Y -180.849,Z 505.472,A 0.000,B 0.000,C 90.000,E1 264.951} C_DIS
LIN {X 0.070,Y -178.897,Z 505.443,A 0.000,B 0.000,C 90.000,E1 259.690} C_DIS
LIN {X -0.026,Y -175.940,Z 505.415,A 0.000,B 0.000,C 90.000,E1 254.629} C_DIS
LIN {X 0.090,Y -175.394,Z 505.410,A 0.000,B 0.000,C 90.000,E1 253.740} C_DIS
LIN {X -0.075,Y -172.163,Z 505.386,A 0.000,B 0.000,C 90.000,E1 249.518} C_DIS
LIN {X -0.036,Y -171.631,Z 505.381,A 0.000,B 0.000,C 90.000,E1 248.646} C_DIS
LIN {X -0.040,Y -167.854,Z 505.357,A 0.000,B 0.000,C 90.000,E1 244.332} C_DIS
LIN {X -0.097,Y -166.586,Z 505.348,A 0.000,B 0.000,C 90.000,E1 242.615} C_DIS
LIN {X 0.037,Y -162.577,Z 505.323,A 0.000,B 0.000,C 90.000,E1 238.201} C_DIS
LIN {X 0.097,Y -161.258,Z 505.314,A 0.000,B 0.000,C 90.000,E1 236.421} C_DIS
LIN {X 0.006,Y -157.260,Z 505.289,A 0.000,B 0.000,C 90.000,E1 232.029} C_DIS
LIN {X -0.068,Y -155.981,Z 505.279,A 0.000,B 0.000,C 90.000,E1 230.275} C_DIS
LIN {X 0.003,Y -152.238,Z 505.254,A 0.000,B 0.000,C 90.000,E1 225.769} C_DIS
LIN {X 0.019,Y -150.478,Z 505.239,A 0.000,B 0.000,C 90.000,E1 223.056} C_DIS
LIN {X -0.052,Y -147.203,Z 505.214,A 0.000,B 0.000,C 90.000,E1 218.543} C_DIS
LIN {X -0.081,Y -145.223,Z 505.194,A 0.000,B 0.000,C 90.000,E1 214.898} C_DIS
LIN {X 0.030,Y -142.351,Z 505.163,A 0.000,B 0.000,C 90.000,E1 209.333} C_DIS
LIN {X -0.043,Y -141.738,Z 505.153,A 0.000,B 0.000,C 90.000,E1 207.513} C_DIS
LIN {X 0.064,Y -139.487,Z 505.117,A 0.000,B 0.000,C 90.000,E1 200.972} C_DIS
LIN {X 0.053,Y -138.988,Z 505.101,A 0.000,B 0.000,C 90.000,E1 198.181} C_DIS
LIN {X 0.014,Y -138.335,Z 505.054,A 0.000,B 0.000,C 90.000,E1 189.792} C_DIS
LIN {X 0.038,Y -139.421,Z 505.008,A 0.000,B 0.000,C 90.000,E1 181.375} C_DIS
LIN {X -0.048,Y -141.341,Z 504.972,A 0.000,B 0.000,C 90.000,E1 174.894} C_DIS
LIN {X 0.069,Y -142.697,Z 504.956,A 0.000,B 0.000,C 90.000,E1 172.064} C_DIS
LIN {X 0.029,Y -145.064,Z 504.930,A 0.000,B 0.000,C 90.000,E1 167.465} C_DIS
LIN {X 0.026,Y -147.689,Z 504.910,A 0.000,B 0.000,C 90.000,E1 163.795} C_DIS
LIN {X -0.083,Y -150.337,Z 504.890,A 0.000,B 0.000,C 90.000,E1 160.188} C_DIS
LIN {X 0.053,Y -154.591,Z 504.865,A 0.000,B 0.000,C 90.000,E1 155.613} C_DIS
LIN {X 0.061,Y -158.129,Z 504.845,A 0.000,B 0.000,C 90.000,E1 152.025} C_DIS
LIN {X 0.020,Y -162.416,Z 504.825,A 0.000,B 0.000,C 90.000,E1 148.486} C_DIS
LIN {X 0.002,Y -166.671,Z 504.805,A 0.000,B 0.000,C 90.000,E1 144.975} C_DIS
LIN {X 0.009,Y -171.678,Z 504.786,A 0.000,B 0.000,C 90.000,E1 141.492} C_DIS
LIN {X -0.081,Y -176.647,Z 504.767,A 0.000,B 0.000,C 90.000,E1 138.081} C_DIS
LIN {X 0.047,Y -180.944,Z 504.753,A 0.000,B 0.000,C 90.000,E1 135.486} C_DIS
LIN {X 0.035,Y -186.364,Z 504.734,A 0.000,B 0.000,C 90.000,E1 132.123} C_DIS
LIN {X -0.024,Y -190.995,Z 504.720,A 0.000,B 0.000,C 90.000,E1 129.644} C_DIS
LIN {X -0.012,Y -192.673,Z 504.715,A 0.000,B 0.000,C 90.000,E1 128.624} C_DIS
LIN {X -0.068,Y -289.705,Z 504.715,A 0.000,B 0.000,C 90.000,E1 128.624} C_DIS
LIN {X -0.082,Y -294.790,Z 504.714,A 0.000,B 0.000,C 90.000,E1 128.463} C_DIS
LIN {X -0.045,Y -296.980,Z 504.713,A 0.000,B 0.000,C 90.000,E1 128.302} C_DIS
LIN {X 0.082,Y -299.983,Z 504.711,A 0.000,B 0.000,C 90.000,E1 127.971} C_DIS
LIN {X 0.060,Y -303.631,Z 504.708,A 0.000,B 0.000,C 90.000,E1 127.397} C_DIS
LIN {X 0.008,Y -305.093,Z 504.706,A 0.000,B 0.000,C 90.000,E1 127.076} C_DIS
LIN {X 0.016,Y -306.248,Z 504.704,A 0.000,B 0.000,C 90.000,E1 126.744} C_DIS
LIN {X -0.061,Y -316.186,Z 504.686,A 0.000,B 0.000,C 90.000,E1 123.499} C_DIS
LIN {X 0.107,Y -326.426,Z 504.670,A 0.000,B 0.000,C 90.000,E1 120.590} C_DIS
LIN {X 0.075,Y -338.015,Z 504.654,A 0.000,B 0.000,C 90.000,E1 117.769} C_DIS
LIN {X -0.092,Y -351.050,Z 504.639,A 0.000,B 0.000,C 90.000,E1 115.027} C_DIS
LIN {X 0.077,Y -363.950,Z 504.626,A 0.000,B 0.000,C 90.000,E1 112.589} C_DIS
LIN {X -0.040,Y -378.184,Z 504.612,A 0.000,B 0.000,C 90.000,E1 110.248} C_DIS
LIN {X -0.067,Y -393.854,Z 504.600,A 0.000,B 0.000,C 90.000,E1 107.946} C_DIS
LIN {X 0.178,Y -411.074,Z 504.587,A 0.000,B 0.000,C 90.000,E1 105.662} C_DIS
LIN {X 0.130,Y -429.972,Z 504.575,A 0.000,B 0.000,C 90.000,E1 103.480} C_DIS
LIN {X 0.072,Y -450.047,Z 504.564,A 0.000,B 0.000,C 90.000,E1 101.422} C_DIS
LIN {X -0.155,Y -470.676,Z 504.553,A 0.000,B 0.000,C 90.000,E1 99.557} C_DIS
LIN {X 0.065,Y -478.555,Z 504.549,A 0.000,B 0.000,C 90.000,E1 98.859} C_DIS
LIN {X 0.200,Y -480.806,Z 504.548,A 0.000,B 0.000,C 90.000,E1 98.624} C_DIS
LIN {X -0.215,Y -482.515,Z 504.547,A 0.000,B 0.000,C 90.000,E1 98.454} C_DIS
LIN {X 0.142,Y -484.001,Z 504.545,A 0.000,B 0.000,C 90.000,E1 98.163} C_DIS
LIN {X -0.048,Y -485.113,Z 504.544,A 0.000,B 0.000,C 90.000,E1 97.936} C_DIS
LIN {X 0.204,Y -486.428,Z 504.541,A 0.000,B 0.000,C 90.000,E1 97.409} C_DIS
LIN {X -0.087,Y -486.718,Z 504.539,A 0.000,B 0.000,C 90.000,E1 96.947} C_DIS
LIN {X 0.112,Y -486.027,Z 504.536,A 0.000,B 0.000,C 90.000,E1 96.429} C_DIS
LIN {X -0.169,Y -484.240,Z 504.533,A 0.000,B 0.000,C 90.000,E1 95.967} C_DIS
LIN {X 0.146,Y -482.831,Z 504.532,A 0.000,B 0.000,C 90.000,E1 95.682} C_DIS
LIN {X 0.160,Y -476.926,Z 504.528,A 0.000,B 0.000,C 90.000,E1 94.935} C_DIS
LIN {X -0.167,Y -462.938,Z 504.518,A 0.000,B 0.000,C 90.000,E1 93.212} C_DIS
LIN {X -0.064,Y -452.045,Z 504.509,A 0.000,B 0.000,C 90.000,E1 91.661} C_DIS
LIN {X -0.072,Y -437.309,Z 504.496,A 0.000,B 0.000,C 90.000,E1 89.312} C_DIS
LIN {X 0.010,Y -427.505,Z 504.487,A 0.000,B 0.000,C 90.000,E1 87.707} C_DIS
LIN {X 0.144,Y -414.632,Z 504.475,A 0.000,B 0.000,C 90.000,E1 85.527} C_DIS
LIN {X 0.080,Y -400.408,Z 504.461,A 0.000,B 0.000,C 90.000,E1 83.053} C_DIS
LIN {X 0.025,Y -391.018,Z 504.452,A 0.000,B 0.000,C 90.000,E1 81.376} C_DIS
LIN {X -0.098,Y -380.028,Z 504.441,A 0.000,B 0.000,C 90.000,E1 79.398} C_DIS
LIN {X -0.015,Y -367.566,Z 504.428,A 0.000,B 0.000,C 90.000,E1 77.061} C_DIS
LIN {X -0.026,Y -357.493,Z 504.417,A 0.000,B 0.000,C 90.000,E1 74.991} C_DIS
LIN {X -0.074,Y -349.551,Z 504.407,A 0.000,B 0.000,C 90.000,E1 73.196} C_DIS
LIN {X 0.085,Y -337.963,Z 504.390,A 0.000,B 0.000,C 90.000,E1 70.115} C_DIS
LIN {X -0.070,Y -326.450,Z 504.371,A 0.000,B 0.000,C 90.000,E1 66.719} C_DIS
LIN {X 0.129,Y -318.517,Z 504.357,A 0.000,B 0.000,C 90.000,E1 64.152} C_DIS
LIN {X -0.169,Y -310.650,Z 504.342,A 0.000,B 0.000,C 90.000,E1 61.641} C_DIS
LIN {X 0.060,Y -302.794,Z 504.328,A 0.000,B 0.000,C 90.000,E1 58.997} C_DIS
LIN {X -0.088,Y -293.253,Z 504.309,A 0.000,B 0.000,C 90.000,E1 55.722} C_DIS
LIN {X -0.035,Y -284.364,Z 504.291,A 0.000,B 0.000,C 90.000,E1 52.351} C_DIS
LIN {X 0.127,Y -278.906,Z 504.279,A 0.000,B 0.000,C 90.000,E1 50.275} C_DIS
LIN {X -0.026,Y -272.970,Z 504.268,A 0.000,B 0.000,C 90.000,E1 48.243} C_DIS
LIN {X -0.003,Y -267.531,Z 504.258,A 0.000,B 0.000,C 90.000,E1 46.500} C_DIS
LIN {X 0.020,Y -259.482,Z 504.245,A 0.000,B 0.000,C 90.000,E1 44.028} C_DIS
LIN {X 0.083,Y -249.196,Z 504.227,A 0.000,B 0.000,C 90.000,E1 40.782} C_DIS
LIN {X -0.046,Y -241.589,Z 504.212,A 0.000,B 0.000,C 90.000,E1 38.257} C_DIS
LIN {X -0.124,Y -233.457,Z 504.196,A 0.000,B 0.000,C 90.000,E1 35.311} C_DIS
LIN {X 0.025,Y -225.992,Z 504.179,A 0.000,B 0.000,C 90.000,E1 32.260} C_DIS
LIN {X 0.005,Y -219.459,Z 504.162,A 0.000,B 0.000,C 90.000,E1 29.205} C_DIS
LIN {X 0.001,Y -213.721,Z 504.145,A 0.000,B 0.000,C 90.000,E1 26.104} C_DIS
LIN {X 0.052,Y -208.938,Z 504.128,A 0.000,B 0.000,C 90.000,E1 22.950} C_DIS
LIN {X -0.064,Y -203.964,Z 504.106,A 0.000,B 0.000,C 90.000,E1 19.014} C_DIS
LIN {X -0.080,Y -199.911,Z 504.083,A 0.000,B 0.000,C 90.000,E1 15.009} C_DIS
LIN {X -0.037,Y -196.417,Z 504.056,A 0.000,B 0.000,C 90.000,E1 10.141} C_DIS
LIN {X -0.071,Y -193.846,Z 504.015,A 0.000,B 0.000,C 90.000,E1 2.808} C_DIS
LIN {X -0.035,Y -195.389,Z 503.961,A 0.000,B 0.000,C 90.000,E1 352.996} C_DIS
LIN {X -0.067,Y -198.342,Z 503.934,A 0.000,B 0.000,C 90.000,E1 348.117} C_DIS
LIN {X 0.017,Y -201.877,Z 503.911,A 0.000,B 0.000,C 90.000,E1 344.047} C_DIS
LIN {X -0.082,Y -206.325,Z 503.889,A 0.000,B 0.000,C 90.000,E1 340.061} C_DIS
LIN {X 0.058,Y -211.577,Z 503.867,A 0.000,B 0.000,C 90.000,E1 336.049} C_DIS
LIN {X -0.060,Y -217.441,Z 503.845,A 0.000,B 0.000,C 90.000,E1 332.153} C_DIS
LIN {X 0.039,Y -223.922,Z 503.824,A 0.000,B 0.000,C 90.000,E1 328.250} C_DIS
LIN {X 0.134,Y -231.083,Z 503.802,A 0.000,B 0.000,C 90.000,E1 324.402} C_DIS
LIN {X 0.111,Y -238.797,Z 503.781,A 0.000,B 0.000,C 90.000,E1 320.642} C_DIS
LIN {X -0.107,Y -247.451,Z 503.761,A 0.000,B 0.000,C 90.000,E1 316.986} C_DIS
LIN {X -0.097,Y -256.313,Z 503.743,A 0.000,B 0.000,C 90.000,E1 313.704} C_DIS
LIN {X 0.097,Y -267.269,Z 503.723,A 0.000,B 0.000,C 90.000,E1 310.092} C_DIS
LIN {X -0.045,Y -279.514,Z 503.703,A 0.000,B 0.000,C 90.000,E1 306.629} C_DIS
LIN {X -0.019,Y -293.026,Z 503.685,A 0.000,B 0.000,C 90.000,E1 303.214} C_DIS
LIN {X 0.032,Y -305.972,Z 503.668,A 0.000,B 0.000,C 90.000,E1 300.207} C_DIS
LIN {X 0.093,Y -321.629,Z 503.650,A 0.000,B 0.000,C 90.000,E1 296.950} C_DIS
LIN {X -0.137,Y -333.975,Z 503.637,A 0.000,B 0.000,C 90.000,E1 294.771} C_DIS
LIN {X -0.065,Y -349.572,Z 503.624,A 0.000,B 0.000,C 90.000,E1 292.280} C_DIS
LIN {X -0.110,Y -369.085,Z 503.609,A 0.000,B 0.000,C 90.000,E1 289.577} C_DIS
LIN {X 0.162,Y -390.506,Z 503.594,A 0.000,B 0.000,C 90.000,E1 286.913} C_DIS
LIN {X 0.079,Y -412.720,Z 503.580,A 0.000,B 0.000,C 90.000,E1 284.426} C_DIS
LIN {X 0.136,Y -425.260,Z 503.573,A 0.000,B 0.000,C 90.000,E1 283.063} C_DIS
LIN {X 0.163,Y -437.557,Z 503.565,A 0.000,B 0.000,C 90.000,E1 281.715} C_DIS
LIN {X 0.135,Y -446.976,Z 503.559,A 0.000,B 0.000,C 90.000,E1 280.658} C_DIS
LIN {X 0.132,Y -455.776,Z 503.553,A 0.000,B 0.000,C 90.000,E1 279.613} C_DIS
LIN {X -0.043,Y -461.720,Z 503.549,A 0.000,B 0.000,C 90.000,E1 278.859} C_DIS
LIN {X -0.175,Y -467.089,Z 503.545,A 0.000,B 0.000,C 90.000,E1 278.106} C_DIS
LIN {X 0.211,Y -471.935,Z 503.541,A 0.000,B 0.000,C 90.000,E1 277.296} C_DIS
LIN {X 0.111,Y -476.248,Z 503.536,A 0.000,B 0.000,C 90.000,E1 276.549} C_DIS
LIN {X 0.108,Y -479.951,Z 503.532,A 0.000,B 0.000,C 90.000,E1 275.796} C_DIS
LIN {X 0.083,Y -483.109,Z 503.528,A 0.000,B 0.000,C 90.000,E1 275.049} C_DIS
LIN {X -0.232,Y -484.853,Z 503.525,A 0.000,B 0.000,C 90.000,E1 274.588} C_DIS
LIN {X -0.089,Y -486.271,Z 503.523,A 0.000,B 0.000,C 90.000,E1 274.073} C_DIS
LIN {X 0.101,Y -487.370,Z 503.520,A 0.000,B 0.000,C 90.000,E1 273.555} C_DIS
LIN {X -0.192,Y -488.165,Z 503.517,A 0.000,B 0.000,C 90.000,E1 273.094} C_DIS
LIN {X -0.018,Y -488.568,Z 503.514,A 0.000,B 0.000,C 90.000,E1 272.579} C_DIS
LIN {X 0.164,Y -488.627,Z 503.512,A 0.000,B 0.000,C 90.000,E1 272.064} C_DIS
LIN {X -0.124,Y -488.317,Z 503.509,A 0.000,B 0.000,C 90.000,E1 271.604} C_DIS
LIN {X 0.061,Y -487.553,Z 503.506,A 0.000,B 0.000,C 90.000,E1 271.088} C_DIS
LIN {X -0.241,Y -486.276,Z 503.503,A 0.000,B 0.000,C 90.000,E1 270.630} C_DIS
LIN {X -0.060,Y -484.517,Z 503.501,A 0.000,B 0.000,C 90.000,E1 270.115} C_DIS
LIN {X 0.112,Y -482.082,Z 503.498,A 0.000,B 0.000,C 90.000,E1 269.599} C_DIS
LIN {X -0.051,Y -480.620,Z 503.496,A 0.000,B 0.000,C 90.000,E1 269.370} C_DIS
LIN {X 0.095,Y -477.028,Z 503.494,A 0.000,B 0.000,C 90.000,E1 268.854} C_DIS
LIN {X -0.075,Y -474.899,Z 503.492,A 0.000,B 0.000,C 90.000,E1 268.625} C_DIS
LIN {X 0.055,Y -469.741,Z 503.490,A 0.000,B 0.000,C 90.000,E1 268.108} C_DIS
LIN {X -0.043,Y -463.827,Z 503.487,A 0.000,B 0.000,C 90.000,E1 267.650} C_DIS
LIN {X -0.122,Y -457.133,Z 503.485,A 0.000,B 0.000,C 90.000,E1 267.249} C_DIS
LIN {X -0.084,Y -450.380,Z 503.483,A 0.000,B 0.000,C 90.000,E1 266.906} C_DIS
LIN {X -0.048,Y -443.453,Z 503.481,A 0.000,B 0.000,C 90.000,E1 266.617} C_DIS
LIN {X -0.106,Y -436.264,Z 503.480,A 0.000,B 0.000,C 90.000,E1 266.388} C_DIS
LIN {X 0.184,Y -428.265,Z 503.479,A 0.000,B 0.000,C 90.000,E1 266.159} C_DIS
LIN {X 0.024,Y -419.013,Z 503.478,A 0.000,B 0.000,C 90.000,E1 266.045} C_DIS
LIN {X -0.049,Y -407.281,Z 503.478,A 0.000,B 0.000,C 90.000,E1 265.988} C_DIS
LIN {X -0.058,Y -180.918,Z 503.478,A 0.000,B 0.000,C 90.000,E1 265.988} C_DIS
LIN {X -0.018,Y -180.848,Z 503.472,A 0.000,B 0.000,C 90.000,E1 264.951} C_DIS
LIN {X 0.059,Y -178.895,Z 503.443,A 0.000,B 0.000,C 90.000,E1 259.690} C_DIS
LIN {X -0.035,Y -175.939,Z 503.415,A 0.000,B 0.000,C 90.000,E1 254.629} C_DIS
LIN {X 0.079,Y -175.390,Z 503.410,A 0.000,B 0.000,C 90.000,E1 253.740} C_DIS
LIN {X -0.085,Y -172.161,Z 503.386,A 0.000,B 0.000,C 90.000,E1 249.518} C_DIS
LIN {X -0.046,Y -171.629,Z 503.381,A 0.000,B 0.000,C 90.000,E1 248.646} C_DIS
LIN {X -0.050,Y -167.851,Z 503.357,A 0.000,B 0.000,C 90.000,E1 244.332} C_DIS
LIN {X 0.041,Y -166.582,Z 503.348,A 0.000,B 0.000,C 90.000,E1 242.564} C_DIS
LIN {X 0.027,Y -162.574,Z 503.323,A 0.000,B 0.000,C 90.000,E1 238.201} C_DIS
LIN {X 0.087,Y -161.255,Z 503.314,A 0.000,B 0.000,C 90.000,E1 236.421} C_DIS
LIN {X -0.003,Y -157.257,Z 503.289,A 0.000,B 0.000,C 90.000,E1 232.029} C_DIS
LIN {X -0.077,Y -155.978,Z 503.279,A 0.000,B 0.000,C 90.000,E1 230.275} C_DIS
LIN {X -0.007,Y -152.235,Z 503.254,A 0.000,B 0.000,C 90.000,E1 225.769} C_DIS
LIN {X 0.010,Y -150.476,Z 503.239,A 0.000,B 0.000,C 90.000,E1 223.056} C_DIS
LIN {X -0.061,Y -147.201,Z 503.214,A 0.000,B 0.000,C 90.000,E1 218.543} C_DIS
LIN {X -0.008,Y -145.221,Z 503.194,A 0.000,B 0.000,C 90.000,E1 214.865} C_DIS
LIN {X 0.020,Y -142.350,Z 503.163,A 0.000,B 0.000,C 90.000,E1 209.333} C_DIS
LIN {X -0.052,Y -141.737,Z 503.153,A 0.000,B 0.000,C 90.000,E1 207.513} C_DIS
LIN {X 0.055,Y -139.486,Z 503.117,A 0.000,B 0.000,C 90.000,E1 200.972} C_DIS
LIN {X 0.044,Y -138.987,Z 503.101,A 0.000,B 0.000,C 90.000,E1 198.181} C_DIS
LIN {X 0.005,Y -138.334,Z 503.054,A 0.000,B 0.000,C 90.000,E1 189.792} C_DIS
LIN {X 0.029,Y -139.422,Z 503.008,A 0.000,B 0.000,C 90.000,E1 181.375} C_DIS
LIN {X -0.057,Y -141.343,Z 502.971,A 0.000,B 0.000,C 90.000,E1 174.894} C_DIS
LIN {X 0.060,Y -142.698,Z 502.956,A 0.000,B 0.000,C 90.000,E1 172.064} C_DIS
LIN {X 0.019,Y -145.066,Z 502.930,A 0.000,B 0.000,C 90.000,E1 167.465} C_DIS
LIN {X 0.016,Y -147.692,Z 502.910,A 0.000,B 0.000,C 90.000,E1 163.795} C_DIS
LIN {X 0.049,Y -150.341,Z 502.890,A 0.000,B 0.000,C 90.000,E1 160.134} C_DIS
LIN {X 0.043,Y -154.595,Z 502.865,A 0.000,B 0.000,C 90.000,E1 155.613} C_DIS
LIN {X 0.050,Y -158.133,Z 502.845,A 0.000,B 0.000,C 90.000,E1 152.025} C_DIS
LIN {X 0.011,Y -162.420,Z 502.825,A 0.000,B 0.000,C 90.000,E1 148.486} C_DIS
LIN {X -0.008,Y -166.676,Z 502.805,A 0.000,B 0.000,C 90.000,E1 144.975} C_DIS
LIN {X -0.001,Y -171.683,Z 502.786,A 0.000,B 0.000,C 90.000,E1 141.492} C_DIS
LIN {X -0.091,Y -176.652,Z 502.767,A 0.000,B 0.000,C 90.000,E1 138.081} C_DIS
LIN {X 0.036,Y -180.949,Z 502.753,A 0.000,B 0.000,C 90.000,E1 135.486} C_DIS
LIN {X 0.024,Y -186.370,Z 502.734,A 0.000,B 0.000,C 90.000,E1 132.123} C_DIS
LIN {X -0.036,Y -191.002,Z 502.720,A 0.000,B 0.000,C 90.000,E1 129.644} C_DIS
LIN {X -0.041,Y -192.749,Z 502.714,A 0.000,B 0.000,C 90.000,E1 128.588} C_DIS
LIN {X 0.129,Y -289.999,Z 502.714,A 0.000,B 0.000,C 90.000,E1 128.543} C_DIS
LIN {X -0.069,Y -292.048,Z 502.714,A 0.000,B 0.000,C 90.000,E1 128.543} C_DIS
LIN {X -0.003,Y -297.039,Z 502.713,A 0.000,B 0.000,C 90.000,E1 128.257} C_DIS
LIN {X 0.066,Y -299.777,Z 502.711,A 0.000,B 0.000,C 90.000,E1 127.971} C_DIS
LIN {X -0.143,Y -303.486,Z 502.708,A 0.000,B 0.000,C 90.000,E1 127.443} C_DIS
LIN {X 0.046,Y -305.000,Z 502.706,A 0.000,B 0.000,C 90.000,E1 127.076} C_DIS
LIN {X 0.053,Y -306.193,Z 502.704,A 0.000,B 0.000,C 90.000,E1 126.744} C_DIS
LIN {X 0.040,Y -317.217,Z 502.684,A 0.000,B 0.000,C 90.000,E1 123.166} C_DIS
LIN {X -0.208,Y -327.600,Z 502.668,A 0.000,B 0.000,C 90.000,E1 120.335} C_DIS
LIN {X 0.092,Y -339.338,Z 502.653,A 0.000,B 0.000,C 90.000,E1 117.462} C_DIS
LIN {X -0.033,Y -352.541,Z 502.637,A 0.000,B 0.000,C 90.000,E1 114.719} C_DIS
LIN {X -0.158,Y -365.600,Z 502.624,A 0.000,B 0.000,C 90.000,E1 112.333} C_DIS
LIN {X 0.107,Y -380.004,Z 502.611,A 0.000,B 0.000,C 90.000,E1 109.939} C_DIS
LIN {X 0.128,Y -395.858,Z 502.598,A 0.000,B 0.000,C 90.000,E1 107.638} C_DIS
LIN {X -0.083,Y -413.277,Z 502.586,A 0.000,B 0.000,C 90.000,E1 105.426} C_DIS
LIN {X -0.086,Y -432.389,Z 502.574,A 0.000,B 0.000,C 90.000,E1 103.244} C_DIS
LIN {X 0.017,Y -452.537,Z 502.562,A 0.000,B 0.000,C 90.000,E1 101.186} C_DIS
LIN {X -0.052,Y -473.230,Z 502.552,A 0.000,B 0.000,C 90.000,E1 99.321} C_DIS
LIN {X 0.095,Y -478.480,Z 502.549,A 0.000,B 0.000,C 90.000,E1 98.859} C_DIS
LIN {X 0.247,Y -480.777,Z 502.548,A 0.000,B 0.000,C 90.000,E1 98.624} C_DIS
LIN {X -0.151,Y -482.518,Z 502.547,A 0.000,B 0.000,C 90.000,E1 98.454} C_DIS
LIN {X 0.205,Y -484.047,Z 502.545,A 0.000,B 0.000,C 90.000,E1 98.163} C_DIS
LIN {X 0.015,Y -485.189,Z 502.544,A 0.000,B 0.000,C 90.000,E1 97.936} C_DIS
LIN {X 0.267,Y -486.557,Z 502.541,A 0.000,B 0.000,C 90.000,E1 97.409} C_DIS
LIN {X -0.023,Y -486.891,Z 502.539,A 0.000,B 0.000,C 90.000,E1 96.947} C_DIS
LIN {X 0.178,Y -486.246,Z 502.536,A 0.000,B 0.000,C 90.000,E1 96.429} C_DIS
LIN {X -0.102,Y -484.516,Z 502.533,A 0.000,B 0.000,C 90.000,E1 95.967} C_DIS
LIN {X 0.213,Y -483.142,Z 502.532,A 0.000,B 0.000,C 90.000,E1 95.682} C_DIS
LIN {X -0.248,Y -477.303,Z 502.528,A 0.000,B 0.000,C 90.000,E1 94.992} C_DIS
LIN {X -0.094,Y -463.272,Z 502.518,A 0.000,B 0.000,C 90.000,E1 93.212} C_DIS
LIN {X 0.014,Y -452.342,Z 502.509,A 0.000,B 0.000,C 90.000,E1 91.661} C_DIS
LIN {X 0.010,Y -437.564,Z 502.496,A 0.000,B 0.000,C 90.000,E1 89.312} C_DIS
LIN {X 0.095,Y -427.760,Z 502.487,A 0.000,B 0.000,C 90.000,E1 87.707} C_DIS
LIN {X -0.181,Y -414.897,Z 502.475,A 0.000,B 0.000,C 90.000,E1 85.584} C_DIS
LIN {X 0.172,Y -400.638,Z 502.462,A 0.000,B 0.000,C 90.000,E1 83.053} C_DIS
LIN {X 0.119,Y -391.256,Z 502.452,A 0.000,B 0.000,C 90.000,E1 81.376} C_DIS
LIN {X -0.003,Y -380.248,Z 502.441,A 0.000,B 0.000,C 90.000,E1 79.398} C_DIS
LIN {X 0.088,Y -369.320,Z 502.430,A 0.000,B 0.000,C 90.000,E1 77.353} C_DIS
LIN {X 0.116,Y -359.047,Z 502.418,A 0.000,B 0.000,C 90.000,E1 75.283} C_DIS
LIN {X 0.026,Y -349.714,Z 502.407,A 0.000,B 0.000,C 90.000,E1 73.196} C_DIS
LIN {X 0.070,Y -336.999,Z 502.388,A 0.000,B 0.000,C 90.000,E1 69.826} C_DIS
LIN {X -0.097,Y -326.549,Z 502.371,A 0.000,B 0.000,C 90.000,E1 66.741} C_DIS
LIN {X -0.056,Y -318.579,Z 502.357,A 0.000,B 0.000,C 90.000,E1 64.204} C_DIS
LIN {X -0.068,Y -310.679,Z 502.342,A 0.000,B 0.000,C 90.000,E1 61.641} C_DIS
LIN {X 0.159,Y -302.813,Z 502.328,A 0.000,B 0.000,C 90.000,E1 58.997} C_DIS
LIN {X 0.009,Y -293.243,Z 502.310,A 0.000,B 0.000,C 90.000,E1 55.722} C_DIS
LIN {X 0.058,Y -284.331,Z 502.291,A 0.000,B 0.000,C 90.000,E1 52.351} C_DIS
LIN {X 0.039,Y -278.861,Z 502.280,A 0.000,B 0.000,C 90.000,E1 50.312} C_DIS
LIN {X 0.062,Y -272.937,Z 502.268,A 0.000,B 0.000,C 90.000,E1 48.243} C_DIS
LIN {X -0.102,Y -267.495,Z 502.258,A 0.000,B 0.000,C 90.000,E1 46.539} C_DIS
LIN {X -0.127,Y -260.617,Z 502.247,A 0.000,B 0.000,C 90.000,E1 44.433} C_DIS
LIN {X 0.146,Y -250.327,Z 502.229,A 0.000,B 0.000,C 90.000,E1 41.148} C_DIS
LIN {X 0.023,Y -241.594,Z 502.213,A 0.000,B 0.000,C 90.000,E1 38.257} C_DIS
LIN {X -0.057,Y -233.452,Z 502.196,A 0.000,B 0.000,C 90.000,E1 35.311} C_DIS
LIN {X -0.031,Y -225.984,Z 502.179,A 0.000,B 0.000,C 90.000,E1 32.291} C_DIS
LIN {X 0.069,Y -219.448,Z 502.162,A 0.000,B 0.000,C 90.000,E1 29.205} C_DIS
LIN {X 0.063,Y -213.711,Z 502.145,A 0.000,B 0.000,C 90.000,E1 26.104} C_DIS
LIN {X 0.111,Y -208.934,Z 502.128,A 0.000,B 0.000,C 90.000,E1 22.950} C_DIS
LIN {X -0.073,Y -203.959,Z 502.106,A 0.000,B 0.000,C 90.000,E1 19.033} C_DIS
LIN {X -0.023,Y -199.876,Z 502.083,A 0.000,B 0.000,C 90.000,E1 15.009} C_DIS
LIN {X 0.017,Y -196.380,Z 502.056,A 0.000,B 0.000,C 90.000,E1 10.141} C_DIS
LIN {X -0.020,Y -193.768,Z 502.016,A 0.000,B 0.000,C 90.000,E1 2.808} C_DIS
LIN {X -0.041,Y -195.266,Z 501.961,A 0.000,B 0.000,C 90.000,E1 352.996} C_DIS
LIN {X -0.036,Y -198.198,Z 501.934,A 0.000,B 0.000,C 90.000,E1 348.105} C_DIS
LIN {X 0.057,Y -201.742,Z 501.911,A 0.000,B 0.000,C 90.000,E1 344.031} C_DIS
LIN {X -0.101,Y -206.183,Z 501.889,A 0.000,B 0.000,C 90.000,E1 340.061} C_DIS
LIN {X 0.034,Y -211.443,Z 501.867,A 0.000,B 0.000,C 90.000,E1 336.049} C_DIS
LIN {X -0.090,Y -217.326,Z 501.845,A 0.000,B 0.000,C 90.000,E1 332.153} C_DIS
LIN {X 0.005,Y -223.799,Z 501.824,A 0.000,B 0.000,C 90.000,E1 328.250} C_DIS
LIN {X 0.095,Y -230.941,Z 501.802,A 0.000,B 0.000,C 90.000,E1 324.402} C_DIS
LIN {X 0.065,Y -238.674,Z 501.781,A 0.000,B 0.000,C 90.000,E1 320.642} C_DIS
LIN {X 0.023,Y -247.372,Z 501.761,A 0.000,B 0.000,C 90.000,E1 316.944} C_DIS
LIN {X -0.152,Y -256.257,Z 501.743,A 0.000,B 0.000,C 90.000,E1 313.704} C_DIS
LIN {X 0.039,Y -267.251,Z 501.723,A 0.000,B 0.000,C 90.000,E1 310.092} C_DIS
LIN {X 0.117,Y -279.510,Z 501.703,A 0.000,B 0.000,C 90.000,E1 306.583} C_DIS
LIN {X -0.084,Y -293.028,Z 501.684,A 0.000,B 0.000,C 90.000,E1 303.214} C_DIS
LIN {X -0.004,Y -307.475,Z 501.666,A 0.000,B 0.000,C 90.000,E1 299.873} C_DIS
LIN {X 0.022,Y -321.660,Z 501.650,A 0.000,B 0.000,C 90.000,E1 296.950} C_DIS
LIN {X 0.092,Y -333.998,Z 501.637,A 0.000,B 0.000,C 90.000,E1 294.719} C_DIS
LIN {X -0.141,Y -349.612,Z 501.624,A 0.000,B 0.000,C 90.000,E1 292.280} C_DIS
LIN {X -0.189,Y -369.095,Z 501.609,A 0.000,B 0.000,C 90.000,E1 289.577} C_DIS
LIN {X 0.079,Y -390.534,Z 501.594,A 0.000,B 0.000,C 90.000,E1 286.913} C_DIS
LIN {X 0.117,Y -415.431,Z 501.579,A 0.000,B 0.000,C 90.000,E1 284.120} C_DIS
LIN {X -0.189,Y -427.838,Z 501.571,A 0.000,B 0.000,C 90.000,E1 282.827} C_DIS
LIN {X -0.091,Y -440.028,Z 501.564,A 0.000,B 0.000,C 90.000,E1 281.478} C_DIS
LIN {X -0.098,Y -449.358,Z 501.558,A 0.000,B 0.000,C 90.000,E1 280.423} C_DIS
LIN {X 0.108,Y -455.890,Z 501.553,A 0.000,B 0.000,C 90.000,E1 279.613} C_DIS
LIN {X -0.067,Y -461.837,Z 501.549,A 0.000,B 0.000,C 90.000,E1 278.859} C_DIS
LIN {X -0.197,Y -467.216,Z 501.545,A 0.000,B 0.000,C 90.000,E1 278.106} C_DIS
LIN {X 0.189,Y -472.086,Z 501.541,A 0.000,B 0.000,C 90.000,E1 277.296} C_DIS
LIN {X 0.091,Y -476.389,Z 501.536,A 0.000,B 0.000,C 90.000,E1 276.549} C_DIS
LIN {X 0.089,Y -480.129,Z 501.532,A 0.000,B 0.000,C 90.000,E1 275.796} C_DIS
LIN {X 0.064,Y -483.251,Z 501.528,A 0.000,B 0.000,C 90.000,E1 275.049} C_DIS
LIN {X 0.234,Y -484.970,Z 501.525,A 0.000,B 0.000,C 90.000,E1 274.531} C_DIS
LIN {X -0.105,Y -486.391,Z 501.523,A 0.000,B 0.000,C 90.000,E1 274.073} C_DIS
LIN {X 0.085,Y -487.516,Z 501.520,A 0.000,B 0.000,C 90.000,E1 273.555} C_DIS
LIN {X -0.207,Y -488.296,Z 501.517,A 0.000,B 0.000,C 90.000,E1 273.094} C_DIS
LIN {X -0.033,Y -488.722,Z 501.514,A 0.000,B 0.000,C 90.000,E1 272.579} C_DIS
LIN {X 0.150,Y -488.778,Z 501.512,A 0.000,B 0.000,C 90.000,E1 272.064} C_DIS
LIN {X -0.136,Y -488.457,Z 501.509,A 0.000,B 0.000,C 90.000,E1 271.604} C_DIS
LIN {X 0.050,Y -487.687,Z 501.506,A 0.000,B 0.000,C 90.000,E1 271.088} C_DIS
LIN {X 0.234,Y -486.422,Z 501.503,A 0.000,B 0.000,C 90.000,E1 270.573} C_DIS
LIN {X -0.070,Y -484.623,Z 501.501,A 0.000,B 0.000,C 90.000,E1 270.115} C_DIS
LIN {X 0.103,Y -482.205,Z 501.498,A 0.000,B 0.000,C 90.000,E1 269.599} C_DIS
LIN {X -0.221,Y -479.031,Z 501.495,A 0.000,B 0.000,C 90.000,E1 269.141} C_DIS
LIN {X -0.083,Y -474.976,Z 501.492,A 0.000,B 0.000,C 90.000,E1 268.625} C_DIS
LIN {X 0.047,Y -469.840,Z 501.490,A 0.000,B 0.000,C 90.000,E1 268.108} C_DIS
LIN {X -0.072,Y -463.896,Z 501.487,A 0.000,B 0.000,C 90.000,E1 267.650} C_DIS
LIN {X -0.160,Y -457.244,Z 501.485,A 0.000,B 0.000,C 90.000,E1 267.249} C_DIS
LIN {X -0.136,Y -450.374,Z 501.483,A 0.000,B 0.000,C 90.000,E1 266.906} C_DIS
LIN {X -0.063,Y -443.588,Z 501.481,A 0.000,B 0.000,C 90.000,E1 266.617} C_DIS
LIN {X -0.159,Y -436.216,Z 501.480,A 0.000,B 0.000,C 90.000,E1 266.388} C_DIS
LIN {X 0.083,Y -427.754,Z 501.479,A 0.000,B 0.000,C 90.000,E1 266.159} C_DIS
LIN {X -0.048,Y -418.459,Z 501.478,A 0.000,B 0.000,C 90.000,E1 266.045} C_DIS
LIN {X -0.034,Y -410.006,Z 501.478,A 0.000,B 0.000,C 90.000,E1 265.988} C_DIS
LIN {X -0.050,Y -180.919,Z 501.478,A 0.000,B 0.000,C 90.000,E1 265.988} C_DIS
LIN {X -0.047,Y -180.883,Z 501.473,A 0.000,B 0.000,C 90.000,E1 265.122} C_DIS
LIN {X 0.012,Y -179.002,Z 501.445,A 0.000,B 0.000,C 90.000,E1 260.038} C_DIS
LIN {X -0.069,Y -178.604,Z 501.440,A 0.000,B 0.000,C 90.000,E1 259.218} C_DIS
LIN {X -0.001,Y -175.656,Z 501.412,A 0.000,B 0.000,C 90.000,E1 254.102} C_DIS
LIN {X 0.005,Y -172.373,Z 501.388,A 0.000,B 0.000,C 90.000,E1 249.826} C_DIS
LIN {X 0.018,Y -171.169,Z 501.378,A 0.000,B 0.000,C 90.000,E1 248.103} C_DIS
LIN {X 0.062,Y -167.465,Z 501.354,A 0.000,B 0.000,C 90.000,E1 243.768} C_DIS
LIN {X -0.004,Y -166.862,Z 501.350,A 0.000,B 0.000,C 90.000,E1 242.922} C_DIS
LIN {X 0.050,Y -162.166,Z 501.320,A 0.000,B 0.000,C 90.000,E1 237.661} C_DIS
LIN {X -0.029,Y -160.727,Z 501.311,A 0.000,B 0.000,C 90.000,E1 235.928} C_DIS
LIN {X -0.050,Y -157.531,Z 501.291,A 0.000,B 0.000,C 90.000,E1 232.396} C_DIS
LIN {X 0.007,Y -155.556,Z 501.276,A 0.000,B 0.000,C 90.000,E1 229.703} C_DIS
LIN {X -0.059,Y -151.847,Z 501.251,A 0.000,B 0.000,C 90.000,E1 225.243} C_DIS
LIN {X -0.044,Y -150.067,Z 501.236,A 0.000,B 0.000,C 90.000,E1 222.528} C_DIS
LIN {X -0.009,Y -146.875,Z 501.211,A 0.000,B 0.000,C 90.000,E1 217.971} C_DIS
LIN {X -0.021,Y -145.460,Z 501.196,A 0.000,B 0.000,C 90.000,E1 215.231} C_DIS
LIN {X 0.020,Y -142.876,Z 501.170,A 0.000,B 0.000,C 90.000,E1 210.620} C_DIS
LIN {X 0.019,Y -141.493,Z 501.150,A 0.000,B 0.000,C 90.000,E1 206.924} C_DIS
LIN {X 0.003,Y -139.385,Z 501.113,A 0.000,B 0.000,C 90.000,E1 200.429} C_DIS
LIN {X -0.008,Y -138.841,Z 501.098,A 0.000,B 0.000,C 90.000,E1 197.638} C_DIS
LIN {X 0.052,Y -138.354,Z 501.056,A 0.000,B 0.000,C 90.000,E1 190.141} C_DIS
LIN {X 0.047,Y -139.519,Z 501.005,A 0.000,B 0.000,C 90.000,E1 180.802} C_DIS
LIN {X -0.011,Y -141.180,Z 500.974,A 0.000,B 0.000,C 90.000,E1 175.241} C_DIS
LIN {X -0.041,Y -142.558,Z 500.958,A 0.000,B 0.000,C 90.000,E1 172.470} C_DIS
LIN {X 0.026,Y -144.839,Z 500.932,A 0.000,B 0.000,C 90.000,E1 167.825} C_DIS
LIN {X 0.012,Y -147.462,Z 500.912,A 0.000,B 0.000,C 90.000,E1 164.157} C_DIS
LIN {X 0.040,Y -150.046,Z 500.892,A 0.000,B 0.000,C 90.000,E1 160.496} C_DIS
LIN {X 0.044,Y -153.387,Z 500.872,A 0.000,B 0.000,C 90.000,E1 156.869} C_DIS
LIN {X -0.050,Y -155.919,Z 500.857,A 0.000,B 0.000,C 90.000,E1 154.204} C_DIS
LIN {X 0.066,Y -159.785,Z 500.837,A 0.000,B 0.000,C 90.000,E1 150.589} C_DIS
LIN {X -0.087,Y -162.024,Z 500.827,A 0.000,B 0.000,C 90.000,E1 148.869} C_DIS
LIN {X 0.026,Y -166.219,Z 500.807,A 0.000,B 0.000,C 90.000,E1 145.308} C_DIS
LIN {X 0.028,Y -171.235,Z 500.788,A 0.000,B 0.000,C 90.000,E1 141.823} C_DIS
LIN {X -0.048,Y -176.122,Z 500.769,A 0.000,B 0.000,C 90.000,E1 138.405} C_DIS
LIN {X 0.068,Y -180.388,Z 500.755,A 0.000,B 0.000,C 90.000,E1 135.810} C_DIS
LIN {X 0.044,Y -185.796,Z 500.736,A 0.000,B 0.000,C 90.000,E1 132.447} C_DIS
LIN {X -0.023,Y -190.413,Z 500.722,A 0.000,B 0.000,C 90.000,E1 129.967} C_DIS
LIN {X -0.019,Y -192.814,Z 500.714,A 0.000,B 0.000,C 90.000,E1 128.543} C_DIS
LIN {X -0.070,Y -290.209,Z 500.714,A 0.000,B 0.000,C 90.000,E1 128.543} C_DIS
LIN {X -0.008,Y -291.590,Z 500.714,A 0.000,B 0.000,C 90.000,E1 128.508} C_DIS
LIN {X 0.027,Y -295.948,Z 500.713,A 0.000,B 0.000,C 90.000,E1 128.302} C_DIS
LIN {X 0.036,Y -299.182,Z 500.711,A 0.000,B 0.000,C 90.000,E1 128.016} C_DIS
LIN {X -0.066,Y -302.855,Z 500.708,A 0.000,B 0.000,C 90.000,E1 127.523} C_DIS
LIN {X 0.122,Y -304.524,Z 500.707,A 0.000,B 0.000,C 90.000,E1 127.156} C_DIS
LIN {X -0.118,Y -305.837,Z 500.705,A 0.000,B 0.000,C 90.000,E1 126.870} C_DIS
LIN {X -0.155,Y -316.888,Z 500.685,A 0.000,B 0.000,C 90.000,E1 123.293} C_DIS
LIN {X 0.026,Y -327.230,Z 500.669,A 0.000,B 0.000,C 90.000,E1 120.384} C_DIS
LIN {X -0.143,Y -338.922,Z 500.653,A 0.000,B 0.000,C 90.000,E1 117.590} C_DIS
LIN {X 0.178,Y -352.078,Z 500.638,A 0.000,B 0.000,C 90.000,E1 114.771} C_DIS
LIN {X 0.043,Y -365.091,Z 500.624,A 0.000,B 0.000,C 90.000,E1 112.386} C_DIS
LIN {X -0.189,Y -379.445,Z 500.611,A 0.000,B 0.000,C 90.000,E1 110.066} C_DIS
LIN {X -0.190,Y -395.244,Z 500.599,A 0.000,B 0.000,C 90.000,E1 107.764} C_DIS
LIN {X 0.084,Y -412.605,Z 500.586,A 0.000,B 0.000,C 90.000,E1 105.481} C_DIS
LIN {X 0.065,Y -431.658,Z 500.574,A 0.000,B 0.000,C 90.000,E1 103.300} C_DIS
LIN {X 0.120,Y -451.785,Z 500.563,A 0.000,B 0.000,C 90.000,E1 101.243} C_DIS
LIN {X 0.005,Y -472.460,Z 500.552,A 0.000,B 0.000,C 90.000,E1 99.378} C_DIS
LIN {X -0.261,Y -480.196,Z 500.548,A 0.000,B 0.000,C 90.000,E1 98.746} C_DIS
LIN {X -0.117,Y -482.116,Z 500.547,A 0.000,B 0.000,C 90.000,E1 98.511} C_DIS
LIN {X 0.238,Y -483.785,Z 500.546,A 0.000,B 0.000,C 90.000,E1 98.219} C_DIS
LIN {X 0.046,Y -485.040,Z 500.544,A 0.000,B 0.000,C 90.000,E1 97.992} C_DIS
LIN {X -0.249,Y -486.585,Z 500.542,A 0.000,B 0.000,C 90.000,E1 97.530} C_DIS
LIN {X 0.005,Y -487.076,Z 500.539,A 0.000,B 0.000,C 90.000,E1 97.004} C_DIS
LIN {X 0.205,Y -486.588,Z 500.536,A 0.000,B 0.000,C 90.000,E1 96.486} C_DIS
LIN {X -0.126,Y -485.043,Z 500.533,A 0.000,B 0.000,C 90.000,E1 96.030} C_DIS
LIN {X 0.241,Y -483.790,Z 500.532,A 0.000,B 0.000,C 90.000,E1 95.739} C_DIS
LIN {X 0.077,Y -482.116,Z 500.531,A 0.000,B 0.000,C 90.000,E1 95.511} C_DIS
LIN {X 0.078,Y -469.927,Z 500.522,A 0.000,B 0.000,C 90.000,E1 94.012} C_DIS
LIN {X 0.049,Y -456.558,Z 500.512,A 0.000,B 0.000,C 90.000,E1 92.236} C_DIS
LIN {X 0.222,Y -444.693,Z 500.502,A 0.000,B 0.000,C 90.000,E1 90.401} C_DIS
LIN {X 0.141,Y -433.301,Z 500.492,A 0.000,B 0.000,C 90.000,E1 88.568} C_DIS
LIN {X -0.192,Y -417.094,Z 500.477,A 0.000,B 0.000,C 90.000,E1 85.927} C_DIS
LIN {X 0.138,Y -404.347,Z 500.465,A 0.000,B 0.000,C 90.000,E1 83.685} C_DIS
LIN {X 0.171,Y -393.403,Z 500.454,A 0.000,B 0.000,C 90.000,E1 81.724} C_DIS
LIN {X 0.088,Y -382.390,Z 500.443,A 0.000,B 0.000,C 90.000,E1 79.746} C_DIS
LIN {X -0.137,Y -369.883,Z 500.430,A 0.000,B 0.000,C 90.000,E1 77.465} C_DIS
LIN {X -0.176,Y -359.522,Z 500.419,A 0.000,B 0.000,C 90.000,E1 75.408} C_DIS
LIN {X 0.114,Y -348.909,Z 500.405,A 0.000,B 0.000,C 90.000,E1 72.960} C_DIS
LIN {X -0.083,Y -335.199,Z 500.385,A 0.000,B 0.000,C 90.000,E1 69.316} C_DIS
LIN {X 0.017,Y -324.845,Z 500.368,A 0.000,B 0.000,C 90.000,E1 66.177} C_DIS
LIN {X 0.013,Y -316.839,Z 500.354,A 0.000,B 0.000,C 90.000,E1 63.640} C_DIS
LIN {X 0.096,Y -308.933,Z 500.339,A 0.000,B 0.000,C 90.000,E1 61.051} C_DIS
LIN {X 0.017,Y -301.077,Z 500.325,A 0.000,B 0.000,C 90.000,E1 58.456} C_DIS
LIN {X -0.183,Y -291.600,Z 500.306,A 0.000,B 0.000,C 90.000,E1 55.182} C_DIS
LIN {X -0.115,Y -284.470,Z 500.291,A 0.000,B 0.000,C 90.000,E1 52.477} C_DIS
LIN {X -0.123,Y -279.023,Z 500.280,A 0.000,B 0.000,C 90.000,E1 50.436} C_DIS
LIN {X 0.115,Y -273.108,Z 500.269,A 0.000,B 0.000,C 90.000,E1 48.324} C_DIS
LIN {X -0.047,Y -267.708,Z 500.259,A 0.000,B 0.000,C 90.000,E1 46.620} C_DIS
LIN {X -0.070,Y -260.850,Z 500.247,A 0.000,B 0.000,C 90.000,E1 44.514} C_DIS
LIN {X 0.018,Y -250.580,Z 500.229,A 0.000,B 0.000,C 90.000,E1 41.272} C_DIS
LIN {X -0.100,Y -241.832,Z 500.213,A 0.000,B 0.000,C 90.000,E1 38.382} C_DIS
LIN {X 0.016,Y -233.657,Z 500.197,A 0.000,B 0.000,C 90.000,E1 35.391} C_DIS
LIN {X -0.143,Y -226.161,Z 500.180,A 0.000,B 0.000,C 90.000,E1 32.418} C_DIS
LIN {X -0.038,Y -219.606,Z 500.163,A 0.000,B 0.000,C 90.000,E1 29.333} C_DIS
LIN {X -0.039,Y -213.854,Z 500.146,A 0.000,B 0.000,C 90.000,E1 26.232} C_DIS
LIN {X 0.018,Y -209.045,Z 500.128,A 0.000,B 0.000,C 90.000,E1 23.078} C_DIS
LIN {X 0.101,Y -204.052,Z 500.106,A 0.000,B 0.000,C 90.000,E1 19.087} C_DIS
LIN {X -0.099,Y -199.919,Z 500.084,A 0.000,B 0.000,C 90.000,E1 15.134} C_DIS
LIN {X -0.013,Y -196.393,Z 500.057,A 0.000,B 0.000,C 90.000,E1 10.254} C_DIS
LIN {X -0.008,Y -193.853,Z 500.021,A 0.000,B 0.000,C 90.000,E1 3.726} C_DIS
LIN {X -0.047,Y -195.145,Z 499.961,A 0.000,B 0.000,C 90.000,E1 352.996} C_DIS
LIN {X -0.047,Y -198.064,Z 499.934,A 0.000,B 0.000,C 90.000,E1 348.105} C_DIS
LIN {X 0.042,Y -201.604,Z 499.911,A 0.000,B 0.000,C 90.000,E1 344.031} C_DIS
LIN {X 0.073,Y -206.036,Z 499.889,A 0.000,B 0.000,C 90.000,E1 340.007} C_DIS
LIN {X 0.009,Y -211.309,Z 499.867,A 0.000,B 0.000,C 90.000,E1 336.049} C_DIS
LIN {X 0.073,Y -217.190,Z 499.845,A 0.000,B 0.000,C 90.000,E1 332.103} C_DIS
LIN {X -0.030,Y -223.678,Z 499.824,A 0.000,B 0.000,C 90.000,E1 328.250} C_DIS
LIN {X 0.055,Y -230.802,Z 499.802,A 0.000,B 0.000,C 90.000,E1 324.402} C_DIS
LIN {X 0.020,Y -238.548,Z 499.781,A 0.000,B 0.000,C 90.000,E1 320.642} C_DIS
LIN {X -0.026,Y -247.279,Z 499.761,A 0.000,B 0.000,C 90.000,E1 316.944} C_DIS
LIN {X -0.036,Y -255.143,Z 499.745,A 0.000,B 0.000,C 90.000,E1 314.028} C_DIS
LIN {X -0.077,Y -266.088,Z 499.725,A 0.000,B 0.000,C 90.000,E1 310.458} C_DIS
LIN {X 0.028,Y -276.936,Z 499.707,A 0.000,B 0.000,C 90.000,E1 307.282} C_DIS
LIN {X -0.020,Y -290.224,Z 499.688,A 0.000,B 0.000,C 90.000,E1 303.865} C_DIS
LIN {X -0.119,Y -304.528,Z 499.670,A 0.000,B 0.000,C 90.000,E1 300.541} C_DIS
LIN {X 0.035,Y -320.034,Z 499.651,A 0.000,B 0.000,C 90.000,E1 297.257} C_DIS
LIN {X 0.027,Y -334.021,Z 499.637,A 0.000,B 0.000,C 90.000,E1 294.719} C_DIS
LIN {X -0.077,Y -349.643,Z 499.624,A 0.000,B 0.000,C 90.000,E1 292.259} C_DIS
LIN {X 0.087,Y -369.104,Z 499.609,A 0.000,B 0.000,C 90.000,E1 289.523} C_DIS
LIN {X -0.139,Y -388.134,Z 499.596,A 0.000,B 0.000,C 90.000,E1 287.221} C_DIS
LIN {X -0.093,Y -412.940,Z 499.580,A 0.000,B 0.000,C 90.000,E1 284.411} C_DIS
LIN {X -0.148,Y -425.618,Z 499.572,A 0.000,B 0.000,C 90.000,E1 283.063} C_DIS
LIN {X -0.062,Y -437.874,Z 499.565,A 0.000,B 0.000,C 90.000,E1 281.715} C_DIS
LIN {X -0.091,Y -447.362,Z 499.559,A 0.000,B 0.000,C 90.000,E1 280.658} C_DIS
LIN {X -0.094,Y -456.166,Z 499.553,A 0.000,B 0.000,C 90.000,E1 279.613} C_DIS
LIN {X 0.188,Y -462.116,Z 499.549,A 0.000,B 0.000,C 90.000,E1 278.803} C_DIS
LIN {X 0.064,Y -467.471,Z 499.545,A 0.000,B 0.000,C 90.000,E1 278.049} C_DIS
LIN {X -0.012,Y -472.354,Z 499.541,A 0.000,B 0.000,C 90.000,E1 277.296} C_DIS
LIN {X -0.055,Y -476.639,Z 499.536,A 0.000,B 0.000,C 90.000,E1 276.543} C_DIS
LIN {X -0.112,Y -480.372,Z 499.532,A 0.000,B 0.000,C 90.000,E1 275.796} C_DIS
LIN {X -0.135,Y -483.480,Z 499.528,A 0.000,B 0.000,C 90.000,E1 275.049} C_DIS
LIN {X 0.036,Y -485.169,Z 499.525,A 0.000,B 0.000,C 90.000,E1 274.531} C_DIS
LIN {X 0.216,Y -486.601,Z 499.522,A 0.000,B 0.000,C 90.000,E1 274.012} C_DIS
LIN {X -0.113,Y -487.694,Z 499.520,A 0.000,B 0.000,C 90.000,E1 273.555} C_DIS
LIN {X 0.083,Y -488.477,Z 499.517,A 0.000,B 0.000,C 90.000,E1 273.037} C_DIS
LIN {X -0.228,Y -488.870,Z 499.514,A 0.000,B 0.000,C 90.000,E1 272.579} C_DIS
LIN {X -0.044,Y -488.920,Z 499.511,A 0.000,B 0.000,C 90.000,E1 272.064} C_DIS
LIN {X 0.158,Y -488.573,Z 499.509,A 0.000,B 0.000,C 90.000,E1 271.547} C_DIS
LIN {X -0.143,Y -487.784,Z 499.506,A 0.000,B 0.000,C 90.000,E1 271.088} C_DIS
LIN {X 0.043,Y -486.511,Z 499.503,A 0.000,B 0.000,C 90.000,E1 270.573} C_DIS
LIN {X 0.224,Y -484.698,Z 499.500,A 0.000,B 0.000,C 90.000,E1 270.057} C_DIS
LIN {X -0.086,Y -482.204,Z 499.498,A 0.000,B 0.000,C 90.000,E1 269.599} C_DIS
LIN {X 0.069,Y -479.001,Z 499.495,A 0.000,B 0.000,C 90.000,E1 269.083} C_DIS
LIN {X 0.205,Y -474.874,Z 499.492,A 0.000,B 0.000,C 90.000,E1 268.568} C_DIS
LIN {X -0.137,Y -469.717,Z 499.489,A 0.000,B 0.000,C 90.000,E1 268.108} C_DIS
LIN {X 0.229,Y -463.740,Z 499.487,A 0.000,B 0.000,C 90.000,E1 267.593} C_DIS
LIN {X 0.152,Y -457.050,Z 499.484,A 0.000,B 0.000,C 90.000,E1 267.192} C_DIS
LIN {X 0.198,Y -450.191,Z 499.483,A 0.000,B 0.000,C 90.000,E1 266.849} C_DIS
LIN {X -0.178,Y -443.338,Z 499.481,A 0.000,B 0.000,C 90.000,E1 266.617} C_DIS
LIN {X 0.166,Y -435.894,Z 499.480,A 0.000,B 0.000,C 90.000,E1 266.331} C_DIS
LIN {X 0.024,Y -427.577,Z 499.479,A 0.000,B 0.000,C 90.000,E1 266.159} C_DIS
LIN {X -0.097,Y -418.106,Z 499.478,A 0.000,B 0.000,C 90.000,E1 266.045} C_DIS
LIN {X -0.072,Y -409.640,Z 499.478,A 0.000,B 0.000,C 90.000,E1 265.988} C_DIS
LIN {X -0.067,Y -180.919,Z 499.478,A 0.000,B 0.000,C 90.000,E1 265.988} C_DIS
LIN {X -0.062,Y -180.882,Z 499.473,A 0.000,B 0.000,C 90.000,E1 265.122} C_DIS
LIN {X -0.003,Y -179.002,Z 499.445,A 0.000,B 0.000,C 90.000,E1 260.038} C_DIS
LIN {X 0.091,Y -178.601,Z 499.440,A 0.000,B 0.000,C 90.000,E1 259.162} C_DIS
LIN {X -0.015,Y -175.653,Z 499.412,A 0.000,B 0.000,C 90.000,E1 254.102} C_DIS
LIN {X -0.010,Y -172.370,Z 499.388,A 0.000,B 0.000,C 90.000,E1 249.826} C_DIS
LIN {X 0.005,Y -171.164,Z 499.378,A 0.000,B 0.000,C 90.000,E1 248.103} C_DIS
LIN {X 0.048,Y -167.461,Z 499.354,A 0.000,B 0.000,C 90.000,E1 243.768} C_DIS
LIN {X -0.019,Y -166.858,Z 499.350,A 0.000,B 0.000,C 90.000,E1 242.922} C_DIS
LIN {X 0.046,Y -162.843,Z 499.325,A 0.000,B 0.000,C 90.000,E1 238.535} C_DIS
LIN {X 0.021,Y -161.526,Z 499.316,A 0.000,B 0.000,C 90.000,E1 236.786} C_DIS
LIN {X 0.061,Y -157.527,Z 499.291,A 0.000,B 0.000,C 90.000,E1 232.351} C_DIS
LIN {X -0.006,Y -155.552,Z 499.276,A 0.000,B 0.000,C 90.000,E1 229.703} C_DIS
LIN {X -0.072,Y -151.843,Z 499.251,A 0.000,B 0.000,C 90.000,E1 225.243} C_DIS
LIN {X -0.058,Y -150.062,Z 499.236,A 0.000,B 0.000,C 90.000,E1 222.528} C_DIS
LIN {X -0.023,Y -146.872,Z 499.211,A 0.000,B 0.000,C 90.000,E1 217.971} C_DIS
LIN {X -0.033,Y -145.457,Z 499.196,A 0.000,B 0.000,C 90.000,E1 215.231} C_DIS
LIN {X 0.080,Y -142.872,Z 499.170,A 0.000,B 0.000,C 90.000,E1 210.590} C_DIS
LIN {X 0.005,Y -141.490,Z 499.150,A 0.000,B 0.000,C 90.000,E1 206.924} C_DIS
LIN {X -0.010,Y -139.385,Z 499.113,A 0.000,B 0.000,C 90.000,E1 200.429} C_DIS
LIN {X -0.021,Y -138.840,Z 499.098,A 0.000,B 0.000,C 90.000,E1 197.638} C_DIS
LIN {X 0.039,Y -138.353,Z 499.056,A 0.000,B 0.000,C 90.000,E1 190.141} C_DIS
LIN {X 0.035,Y -139.520,Z 499.005,A 0.000,B 0.000,C 90.000,E1 180.802} C_DIS
LIN {X -0.024,Y -141.182,Z 498.974,A 0.000,B 0.000,C 90.000,E1 175.241} C_DIS
LIN {X -0.054,Y -142.561,Z 498.958,A 0.000,B 0.000,C 90.000,E1 172.470} C_DIS
LIN {X 0.013,Y -144.842,Z 498.932,A 0.000,B 0.000,C 90.000,E1 167.825} C_DIS
LIN {X -0.001,Y -147.466,Z 498.912,A 0.000,B 0.000,C 90.000,E1 164.157} C_DIS
LIN {X 0.026,Y -150.050,Z 498.892,A 0.000,B 0.000,C 90.000,E1 160.496} C_DIS
LIN {X 0.030,Y -153.393,Z 498.872,A 0.000,B 0.000,C 90.000,E1 156.869} C_DIS
LIN {X 0.078,Y -155.924,Z 498.857,A 0.000,B 0.000,C 90.000,E1 154.152} C_DIS
LIN {X 0.052,Y -159.790,Z 498.837,A 0.000,B 0.000,C 90.000,E1 150.589} C_DIS
LIN {X 0.038,Y -162.030,Z 498.827,A 0.000,B 0.000,C 90.000,E1 148.820} C_DIS
LIN {X 0.012,Y -166.226,Z 498.807,A 0.000,B 0.000,C 90.000,E1 145.308} C_DIS
LIN {X 0.013,Y -171.242,Z 498.788,A 0.000,B 0.000,C 90.000,E1 141.823} C_DIS
LIN {X -0.064,Y -176.129,Z 498.769,A 0.000,B 0.000,C 90.000,E1 138.405} C_DIS
LIN {X 0.052,Y -180.396,Z 498.755,A 0.000,B 0.000,C 90.000,E1 135.810} C_DIS
LIN {X 0.029,Y -185.804,Z 498.736,A 0.000,B 0.000,C 90.000,E1 132.447} C_DIS
LIN {X 0.083,Y -190.422,Z 498.722,A 0.000,B 0.000,C 90.000,E1 129.930} C_DIS
LIN {X -0.026,Y -192.878,Z 498.714,A 0.000,B 0.000,C 90.000,E1 128.508} C_DIS
LIN {X 0.152,Y -289.767,Z 498.714,A 0.000,B 0.000,C 90.000,E1 128.463} C_DIS
LIN {X 0.049,Y -291.366,Z 498.714,A 0.000,B 0.000,C 90.000,E1 128.463} C_DIS
LIN {X 0.004,Y -295.480,Z 498.713,A 0.000,B 0.000,C 90.000,E1 128.302} C_DIS
LIN {X 0.148,Y -298.672,Z 498.711,A 0.000,B 0.000,C 90.000,E1 128.016} C_DIS
LIN {X -0.011,Y -302.371,Z 498.709,A 0.000,B 0.000,C 90.000,E1 127.569} C_DIS
LIN {X -0.010,Y -304.170,Z 498.707,A 0.000,B 0.000,C 90.000,E1 127.237} C_DIS
LIN {X 0.177,Y -305.580,Z 498.705,A 0.000,B 0.000,C 90.000,E1 126.870} C_DIS
LIN {X -0.023,Y -307.621,Z 498.701,A 0.000,B 0.000,C 90.000,E1 126.251} C_DIS
LIN {X -0.053,Y -317.766,Z 498.683,A 0.000,B 0.000,C 90.000,E1 123.007} C_DIS
LIN {X -0.011,Y -328.226,Z 498.667,A 0.000,B 0.000,C 90.000,E1 120.129} C_DIS
LIN {X 0.003,Y -340.051,Z 498.652,A 0.000,B 0.000,C 90.000,E1 117.308} C_DIS
LIN {X 0.205,Y -353.343,Z 498.636,A 0.000,B 0.000,C 90.000,E1 114.515} C_DIS
LIN {X -0.039,Y -366.491,Z 498.623,A 0.000,B 0.000,C 90.000,E1 112.153} C_DIS
LIN {X -0.101,Y -380.988,Z 498.610,A 0.000,B 0.000,C 90.000,E1 109.812} C_DIS
LIN {X -0.067,Y -396.944,Z 498.597,A 0.000,B 0.000,C 90.000,E1 107.511} C_DIS
LIN {X 0.132,Y -414.474,Z 498.585,A 0.000,B 0.000,C 90.000,E1 105.245} C_DIS
LIN {X 0.188,Y -433.679,Z 498.573,A 0.000,B 0.000,C 90.000,E1 103.063} C_DIS
LIN {X -0.141,Y -453.866,Z 498.561,A 0.000,B 0.000,C 90.000,E1 101.074} C_DIS
LIN {X -0.124,Y -474.594,Z 498.551,A 0.000,B 0.000,C 90.000,E1 99.208} C_DIS
LIN {X 0.046,Y -479.809,Z 498.549,A 0.000,B 0.000,C 90.000,E1 98.746} C_DIS
LIN {X 0.188,Y -481.869,Z 498.547,A 0.000,B 0.000,C 90.000,E1 98.511} C_DIS
LIN {X 0.064,Y -483.650,Z 498.546,A 0.000,B 0.000,C 90.000,E1 98.276} C_DIS
LIN {X -0.130,Y -484.988,Z 498.545,A 0.000,B 0.000,C 90.000,E1 98.049} C_DIS
LIN {X 0.056,Y -486.661,Z 498.542,A 0.000,B 0.000,C 90.000,E1 97.530} C_DIS
LIN {X -0.234,Y -487.260,Z 498.539,A 0.000,B 0.000,C 90.000,E1 97.068} C_DIS
LIN {X -0.029,Y -486.880,Z 498.536,A 0.000,B 0.000,C 90.000,E1 96.549} C_DIS
LIN {X 0.179,Y -485.459,Z 498.534,A 0.000,B 0.000,C 90.000,E1 96.030} C_DIS
LIN {X 0.064,Y -484.283,Z 498.532,A 0.000,B 0.000,C 90.000,E1 95.796} C_DIS
LIN {X -0.099,Y -482.710,Z 498.531,A 0.000,B 0.000,C 90.000,E1 95.568} C_DIS
LIN {X 0.066,Y -472.559,Z 498.524,A 0.000,B 0.000,C 90.000,E1 94.302} C_DIS
LIN {X -0.128,Y -460.787,Z 498.516,A 0.000,B 0.000,C 90.000,E1 92.808} C_DIS
LIN {X -0.085,Y -450.090,Z 498.507,A 0.000,B 0.000,C 90.000,E1 91.260} C_DIS
LIN {X 0.125,Y -437.009,Z 498.495,A 0.000,B 0.000,C 90.000,E1 89.141} C_DIS
LIN {X 0.033,Y -423.919,Z 498.483,A 0.000,B 0.000,C 90.000,E1 87.020} C_DIS
LIN {X 0.026,Y -412.737,Z 498.473,A 0.000,B 0.000,C 90.000,E1 85.122} C_DIS
LIN {X -0.079,Y -398.517,Z 498.459,A 0.000,B 0.000,C 90.000,E1 82.648} C_DIS
LIN {X -0.164,Y -389.087,Z 498.450,A 0.000,B 0.000,C 90.000,E1 80.971} C_DIS
LIN {X 0.121,Y -378.089,Z 498.439,A 0.000,B 0.000,C 90.000,E1 78.926} C_DIS
LIN {X 0.169,Y -361.312,Z 498.421,A 0.000,B 0.000,C 90.000,E1 75.700} C_DIS
LIN {X 0.094,Y -349.239,Z 498.406,A 0.000,B 0.000,C 90.000,E1 73.015} C_DIS
LIN {X 0.111,Y -335.462,Z 498.385,A 0.000,B 0.000,C 90.000,E1 69.337} C_DIS
LIN {X 0.023,Y -325.069,Z 498.368,A 0.000,B 0.000,C 90.000,E1 66.230} C_DIS
LIN {X 0.030,Y -317.012,Z 498.354,A 0.000,B 0.000,C 90.000,E1 63.691} C_DIS
LIN {X -0.026,Y -309.079,Z 498.340,A 0.000,B 0.000,C 90.000,E1 61.129} C_DIS
LIN {X -0.104,Y -301.199,Z 498.325,A 0.000,B 0.000,C 90.000,E1 58.535} C_DIS
LIN {X 0.105,Y -291.695,Z 498.307,A 0.000,B 0.000,C 90.000,E1 55.182} C_DIS
LIN {X 0.167,Y -284.529,Z 498.292,A 0.000,B 0.000,C 90.000,E1 52.477} C_DIS
LIN {X 0.156,Y -279.075,Z 498.280,A 0.000,B 0.000,C 90.000,E1 50.436} C_DIS
LIN {X 0.003,Y -273.153,Z 498.269,A 0.000,B 0.000,C 90.000,E1 48.405} C_DIS
LIN {X -0.039,Y -268.898,Z 498.261,A 0.000,B 0.000,C 90.000,E1 47.025} C_DIS
LIN {X 0.099,Y -263.271,Z 498.251,A 0.000,B 0.000,C 90.000,E1 45.243} C_DIS
LIN {X 0.024,Y -255.203,Z 498.238,A 0.000,B 0.000,C 90.000,E1 42.771} C_DIS
LIN {X -0.011,Y -246.294,Z 498.222,A 0.000,B 0.000,C 90.000,E1 39.886} C_DIS
LIN {X -0.060,Y -235.753,Z 498.201,A 0.000,B 0.000,C 90.000,E1 36.217} C_DIS
LIN {X -0.045,Y -228.048,Z 498.184,A 0.000,B 0.000,C 90.000,E1 33.214} C_DIS
LIN {X 0.100,Y -221.263,Z 498.168,A 0.000,B 0.000,C 90.000,E1 30.129} C_DIS
LIN {X -0.051,Y -215.290,Z 498.150,A 0.000,B 0.000,C 90.000,E1 27.078} C_DIS
LIN {X -0.058,Y -210.221,Z 498.133,A 0.000,B 0.000,C 90.000,E1 23.951} C_DIS
LIN {X -0.056,Y -205.010,Z 498.111,A 0.000,B 0.000,C 90.000,E1 19.993} C_DIS
LIN {X 0.024,Y -200.670,Z 498.089,A 0.000,B 0.000,C 90.000,E1 15.969} C_DIS
LIN {X -0.010,Y -196.853,Z 498.062,A 0.000,B 0.000,C 90.000,E1 11.130} C_DIS
LIN {X 0.065,Y -193.986,Z 498.026,A 0.000,B 0.000,C 90.000,E1 4.588} C_DIS
LIN {X -0.052,Y -195.024,Z 497.961,A 0.000,B 0.000,C 90.000,E1 352.996} C_DIS
LIN {X -0.057,Y -197.938,Z 497.934,A 0.000,B 0.000,C 90.000,E1 348.105} C_DIS
LIN {X 0.028,Y -201.463,Z 497.911,A 0.000,B 0.000,C 90.000,E1 344.031} C_DIS
LIN {X 0.054,Y -205.885,Z 497.889,A 0.000,B 0.000,C 90.000,E1 340.007} C_DIS
LIN {X -0.014,Y -211.172,Z 497.867,A 0.000,B 0.000,C 90.000,E1 336.049} C_DIS
LIN {X 0.043,Y -217.053,Z 497.845,A 0.000,B 0.000,C 90.000,E1 332.103} C_DIS
LIN {X -0.064,Y -223.556,Z 497.824,A 0.000,B 0.000,C 90.000,E1 328.250} C_DIS
LIN {X 0.016,Y -230.675,Z 497.802,A 0.000,B 0.000,C 90.000,E1 324.402} C_DIS
LIN {X -0.025,Y -238.429,Z 497.781,A 0.000,B 0.000,C 90.000,E1 320.642} C_DIS
LIN {X 0.092,Y -247.187,Z 497.761,A 0.000,B 0.000,C 90.000,E1 316.905} C_DIS
LIN {X -0.090,Y -255.075,Z 497.744,A 0.000,B 0.000,C 90.000,E1 314.028} C_DIS
LIN {X -0.134,Y -266.052,Z 497.725,A 0.000,B 0.000,C 90.000,E1 310.458} C_DIS
LIN {X -0.032,Y -276.926,Z 497.707,A 0.000,B 0.000,C 90.000,E1 307.282} C_DIS
LIN {X 0.077,Y -290.225,Z 497.688,A 0.000,B 0.000,C 90.000,E1 303.833} C_DIS
LIN {X -0.031,Y -304.533,Z 497.669,A 0.000,B 0.000,C 90.000,E1 300.512} C_DIS
LIN {X -0.104,Y -318.426,Z 497.653,A 0.000,B 0.000,C 90.000,E1 297.590} C_DIS
LIN {X -0.014,Y -332.222,Z 497.639,A 0.000,B 0.000,C 90.000,E1 295.027} C_DIS
LIN {X 0.153,Y -347.637,Z 497.625,A 0.000,B 0.000,C 90.000,E1 292.514} C_DIS
LIN {X 0.061,Y -366.852,Z 497.610,A 0.000,B 0.000,C 90.000,E1 289.812} C_DIS
LIN {X -0.221,Y -388.150,Z 497.595,A 0.000,B 0.000,C 90.000,E1 287.221} C_DIS
LIN {X -0.155,Y -412.947,Z 497.580,A 0.000,B 0.000,C 90.000,E1 284.411} C_DIS
LIN {X -0.117,Y -425.530,Z 497.572,A 0.000,B 0.000,C 90.000,E1 283.063} C_DIS
LIN {X -0.048,Y -437.880,Z 497.565,A 0.000,B 0.000,C 90.000,E1 281.715} C_DIS
LIN {X -0.077,Y -447.400,Z 497.559,A 0.000,B 0.000,C 90.000,E1 280.658} C_DIS
LIN {X 0.119,Y -454.126,Z 497.555,A 0.000,B 0.000,C 90.000,E1 279.849} C_DIS
LIN {X -0.075,Y -460.284,Z 497.550,A 0.000,B 0.000,C 90.000,E1 279.095} C_DIS
LIN {X 0.080,Y -467.576,Z 497.545,A 0.000,B 0.000,C 90.000,E1 278.049} C_DIS
LIN {X 0.005,Y -472.466,Z 497.541,A 0.000,B 0.000,C 90.000,E1 277.296} C_DIS
LIN {X -0.091,Y -476.749,Z 497.536,A 0.000,B 0.000,C 90.000,E1 276.549} C_DIS
LIN {X -0.092,Y -480.460,Z 497.532,A 0.000,B 0.000,C 90.000,E1 275.796} C_DIS
LIN {X -0.115,Y -483.605,Z 497.528,A 0.000,B 0.000,C 90.000,E1 275.049} C_DIS
LIN {X 0.057,Y -485.330,Z 497.525,A 0.000,B 0.000,C 90.000,E1 274.531} C_DIS
LIN {X 0.238,Y -486.723,Z 497.522,A 0.000,B 0.000,C 90.000,E1 274.012} C_DIS
LIN {X -0.090,Y -487.847,Z 497.520,A 0.000,B 0.000,C 90.000,E1 273.555} C_DIS
LIN {X 0.107,Y -488.622,Z 497.517,A 0.000,B 0.000,C 90.000,E1 273.037} C_DIS
LIN {X -0.204,Y -489.018,Z 497.514,A 0.000,B 0.000,C 90.000,E1 272.579} C_DIS
LIN {X -0.019,Y -489.075,Z 497.511,A 0.000,B 0.000,C 90.000,E1 272.064} C_DIS
LIN {X 0.184,Y -488.735,Z 497.509,A 0.000,B 0.000,C 90.000,E1 271.547} C_DIS
LIN {X -0.116,Y -487.950,Z 497.506,A 0.000,B 0.000,C 90.000,E1 271.088} C_DIS
LIN {X 0.071,Y -486.690,Z 497.503,A 0.000,B 0.000,C 90.000,E1 270.573} C_DIS
LIN {X -0.232,Y -484.845,Z 497.500,A 0.000,B 0.000,C 90.000,E1 270.115} C_DIS
LIN {X -0.056,Y -482.402,Z 497.498,A 0.000,B 0.000,C 90.000,E1 269.599} C_DIS
LIN {X 0.100,Y -479.161,Z 497.495,A 0.000,B 0.000,C 90.000,E1 269.083} C_DIS
LIN {X -0.238,Y -475.054,Z 497.492,A 0.000,B 0.000,C 90.000,E1 268.625} C_DIS
LIN {X -0.106,Y -469.892,Z 497.489,A 0.000,B 0.000,C 90.000,E1 268.108} C_DIS
